KUKA KRL program: MyProgram_180().src

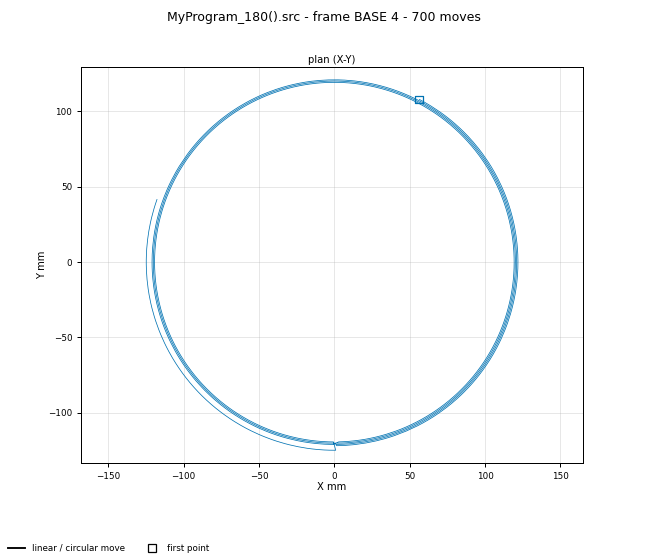
[picture p0: tool path of MyProgram_180().src in frame BASE 4, 700 of 700 moves have a stored position in this frame; points joined in program order, loops and branches not executed]
&ACCESS RVP
&REL 1
&PARAM TEMPLATE = C:\KRC\Roboter\Template\vorgabe
&PARAM EDITMASK = *
DEF MyProgram_180()
; ---- Setting reference (Base) ----
$BASE = BASE_DATA[4]

; --------------------------
; ---- Setting tool (TCP) ----
$TOOL = TOOL_DATA[3]
; --------------------------

$VEL.CP = VEL_APROX_PRINT
Startdeposition()
$VEL.CP = VEL_PRINT
LIN {X 56.4731,Y 107.9839,Z 132,A 57.7826,B 24.9435,C -1.7366,E1 25.0755,E2 388.3875} C_DIS
LIN {X 60.1294,Y 105.9923,Z 132,A 56.1238,B 24.9427,C -1.7481,E1 25.0795,E2 390.0143} C_DIS
LIN {X 64.0212,Y 103.6878,Z 132,A 53.6842,B 24.9439,C -1.7299,E1 25.0854,E2 392.4894} C_DIS
LIN {X 70.1878,Y 99.6172,Z 132,A 50.2313,B 24.9442,C -1.7251,E1 25.0934,E2 395.942} C_DIS
LIN {X 73.4213,Y 97.2579,Z 132,A 48.296,B 24.9446,C -1.7192,E1 25.0977,E2 397.8843} C_DIS
LIN {X 77.0237,Y 94.4306,Z 132,A 46.2185,B 24.9446,C -1.7188,E1 25.1023,E2 399.9551} C_DIS
LIN {X 80.294,Y 91.6663,Z 132,A 44.3805,B 24.9443,C -1.7233,E1 25.1061,E2 401.7753} C_DIS
LIN {X 83.0267,Y 89.1984,Z 132,A 42.6386,B 24.9446,C -1.7192,E1 25.1097,E2 403.5198} C_DIS
LIN {X 85.7566,Y 86.578,Z 132,A 40.7263,B 24.9453,C -1.7089,E1 25.1136,E2 405.4483} C_DIS
LIN {X 88.8179,Y 83.4346,Z 132,A 38.6725,B 24.9455,C -1.7048,E1 25.1175,E2 407.5031} C_DIS
LIN {X 92.0346,Y 79.8719,Z 132,A 36.4485,B 24.9458,C -1.7012,E1 25.1217,E2 409.7257} C_DIS
LIN {X 95.6699,Y 75.4792,Z 132,A 33.745,B 24.9462,C -1.6936,E1 25.1264,E2 412.4344} C_DIS
LIN {X 98.202,Y 72.1549,Z 132,A 31.8136,B 24.9465,C -1.6903,E1 25.1297,E2 414.3644} C_DIS
LIN {X 102.2261,Y 66.3297,Z 132,A 28.5147,B 24.9469,C -1.6831,E1 25.1349,E2 417.664} C_DIS
LIN {X 104.0153,Y 63.4873,Z 132,A 26.4897,B 24.9485,C -1.6571,E1 25.1379,E2 419.7401} C_DIS
LIN {X 106.1427,Y 59.8631,Z 132,A 24.9613,B 24.9475,C -1.6736,E1 25.1399,E2 421.2217} C_DIS
LIN {X 108.2856,Y 55.8944,Z 132,A 22.9017,B 24.9477,C -1.6706,E1 25.1426,E2 423.2774} C_DIS
LIN {X 110.9683,Y 50.3551,Z 132,A 20.0051,B 24.9482,C -1.6622,E1 25.1461,E2 426.1783} C_DIS
LIN {X 112.7882,Y 46.1367,Z 132,A 17.4555,B 24.9498,C -1.6366,E1 25.1489,E2 428.774} C_DIS
LIN {X 114.2155,Y 42.4817,Z 132,A 15.9852,B 24.949,C -1.6496,E1 25.1503,E2 430.2057} C_DIS
LIN {X 115.6712,Y 38.3389,Z 132,A 13.9725,B 24.9492,C -1.6459,E1 25.1521,E2 432.2157} C_DIS
LIN {X 116.887,Y 34.4575,Z 132,A 11.9721,B 24.9499,C -1.6356,E1 25.1537,E2 434.2289} C_DIS
LIN {X 118.1425,Y 29.8669,Z 132,A 9.3487,B 24.9515,C -1.6096,E1 25.1556,E2 436.8985} C_DIS
LIN {X 119.1512,Y 25.5527,Z 132,A 7.3765,B 24.9515,C -1.6085,E1 25.1568,E2 438.8619} C_DIS
LIN {X 119.9017,Y 21.7572,Z 132,A 5.7778,B 24.9512,C -1.6136,E1 25.1576,E2 440.4392} C_DIS
LIN {X 120.553,Y 17.8008,Z 132,A 3.3375,B 24.9532,C -1.5801,E1 25.1586,E2 442.944} C_DIS
LIN {X 121.2462,Y 12.2184,Z 132,A 0.9458,B 24.953,C -1.584,E1 25.1592,E2 445.3124} C_DIS
LIN {X 121.6093,Y 7.7983,Z 132,A -0.5381,B 24.9516,C -1.6071,E1 25.1595,E2 446.7331} C_DIS
LIN {X 121.7541,Y 5.0713,Z 132,A -2.4124,B 24.9536,C -1.5735,E1 25.1598,E2 448.6753} C_DIS
LIN {X 121.8578,Y 0.5482,Z 132,A -3.7742,B 24.9518,C -1.6047,E1 25.1598,E2 449.9557} C_DIS
LIN {X 121.787,Y -4.1979,Z 132,A -6.1962,B 24.9528,C -1.5878,E1 25.1597,E2 452.4031} C_DIS
LIN {X 121.5815,Y -8.2299,Z 132,A -8.1191,B 24.9532,C -1.5803,E1 25.1593,E2 454.3322} C_DIS
LIN {X 121.104,Y -13.5503,Z 132,A -11.226,B 24.9554,C -1.5425,E1 25.1584,E2 457.5097} C_DIS
LIN {X 120.4386,Y -18.5544,Z 132,A -12.6686,B 24.9532,C -1.5811,E1 25.1579,E2 458.853} C_DIS
LIN {X 119.981,Y -21.319,Z 132,A -14.6634,B 24.9554,C -1.5429,E1 25.1569,E2 460.9259} C_DIS
LIN {X 119.1633,Y -25.4976,Z 132,A -16.7801,B 24.9561,C -1.5307,E1 25.1556,E2 463.0591} C_DIS
LIN {X 118.136,Y -29.8926,Z 132,A -18.3594,B 24.9549,C -1.5509,E1 25.1546,E2 464.5818} C_DIS
LIN {X 116.8997,Y -34.4146,Z 132,A -21.4806,B 24.9579,C -1.4984,E1 25.1521,E2 467.8089} C_DIS
LIN {X 114.889,Y -40.6276,Z 132,A -23.6416,B 24.9559,C -1.5336,E1 25.1502,E2 469.8748} C_DIS
LIN {X 113.2694,Y -44.9444,Z 132,A -25.6739,B 24.9559,C -1.5336,E1 25.1482,E2 471.8959} C_DIS
LIN {X 110.7217,Y -50.8989,Z 132,A -28.8215,B 24.9568,C -1.519,E1 25.1446,E2 475.0605} C_DIS
LIN {X 109.2594,Y -53.9659,Z 132,A -30.6777,B 24.9578,C -1.5013,E1 25.1423,E2 476.9486} C_DIS
LIN {X 107.6556,Y -57.0968,Z 132,A -32.5414,B 24.9586,C -1.486,E1 25.1398,E2 478.8386} C_DIS
LIN {X 105.4079,Y -61.1478,Z 132,A -34.1894,B 24.9575,C -1.5057,E1 25.1376,E2 480.4314} C_DIS
LIN {X 103.2812,Y -64.676,Z 132,A -36.1228,B 24.9578,C -1.5003,E1 25.1348,E2 482.3679} C_DIS
LIN {X 100.9382,Y -68.274,Z 132,A -38.0879,B 24.958,C -1.4972,E1 25.1318,E2 484.3305} C_DIS
LIN {X 98.55,Y -71.6776,Z 132,A -40.0435,B 24.9583,C -1.4917,E1 25.1286,E2 486.2896} C_DIS
LIN {X 96.0385,Y -75.0101,Z 132,A -42.2663,B 24.9593,C -1.4734,E1 25.1247,E2 488.545} C_DIS
LIN {X 93.9447,Y -77.6163,Z 132,A -43.566,B 24.9588,C -1.4826,E1 25.1225,E2 489.8168} C_DIS
LIN {X 91.9011,Y -80.0264,Z 132,A -45.4055,B 24.96,C -1.4613,E1 25.1191,E2 491.6985} C_DIS
LIN {X 89.3899,Y -82.8206,Z 132,A -47.373,B 24.9608,C -1.4469,E1 25.1153,E2 493.6911} C_DIS
LIN {X 86.0477,Y -86.2879,Z 132,A -49.0581,B 24.9595,C -1.4697,E1 25.1121,E2 495.3154} C_DIS
LIN {X 83.8181,Y -88.4552,Z 132,A -50.9541,B 24.9609,C -1.4448,E1 25.1081,E2 497.2622} C_DIS
LIN {X 80.6989,Y -91.31,Z 132,A -52.893,B 24.961,C -1.4426,E1 25.1041,E2 499.1988} C_DIS
LIN {X 77.6217,Y -93.9402,Z 132,A -54.3862,B 24.9602,C -1.4583,E1 25.101,E2 500.6491} C_DIS
LIN {X 74.3584,Y -96.5433,Z 132,A -57.188,B 24.9626,C -1.4132,E1 25.0946,E2 503.547} C_DIS
LIN {X 69.3835,Y -100.1788,Z 132,A -59.2103,B 24.9606,C -1.4496,E1 25.0902,E2 505.4765} C_DIS
LIN {X 66.0306,Y -102.4196,Z 132,A -61.1258,B 24.9609,C -1.4449,E1 25.0857,E2 507.3968} C_DIS
LIN {X 62.3586,Y -104.6957,Z 132,A -63.1483,B 24.9611,C -1.4414,E1 25.0808,E2 509.4211} C_DIS
LIN {X 58.664,Y -106.8099,Z 132,A -65.125,B 24.9612,C -1.439,E1 25.076,E2 511.3977} C_DIS
LIN {X 55.147,Y -108.6664,Z 132,A -66.7851,B 24.9608,C -1.446,E1 25.072,E2 513.0367} C_DIS
LIN {X 47.6474,Y -112.1587,Z 132,A -70.8114,B 24.9615,C -1.4332,E1 25.0617,E2 517.083} C_DIS
LIN {X 39.8361,Y -115.1649,Z 132,A -74.7717,B 24.9619,C -1.4265,E1 25.0513,E2 521.0506} C_DIS
LIN {X 35.9115,Y -116.4481,Z 132,A -76.6767,B 24.9619,C -1.4259,E1 25.0463,E2 522.9535} C_DIS
LIN {X 33.0929,Y -117.2805,Z 132,A -78.8349,B 24.9639,C -1.3875,E1 25.0402,E2 525.1992} C_DIS
LIN {X 27.7021,Y -118.6696,Z 132,A -80.6741,B 24.9621,C -1.4217,E1 25.0355,E2 526.9546} C_DIS
LIN {X 20.9444,Y -120.0462,Z 132,A -83.8401,B 24.9621,C -1.4226,E1 25.0268,E2 530.1149} C_DIS
LIN {X 13.1586,Y -121.1476,Z 132,A -87.6463,B 24.9625,C -1.4149,E1 25.0162,E2 533.936} C_DIS
LIN {X 7.5514,Y -121.625,Z 132,A -90.2781,B 24.9625,C -1.4143,E1 25.0089,E2 536.568} C_DIS
LIN {X 1.6031,Y -121.8492,Z 132,A -93.0648,B 24.9625,C -1.4139,E1 25.0011,E2 539.3549} C_DIS
LIN {X 1.6031,Y -121.8492,Z 132,A -93.0648,B 24.9625,C -1.4139,E1 25.0011,E2 539.3549} C_DIS
Enddeposition()
LIN {X 0.8619,Y -121.0153,Z 132,A -93.2429,B 24.9613,C -1.4367,E1 25.0008,E2 539.4791} C_DIS
Startdeposition()
$VEL.CP = VEL_PRINT
LIN {X 6.3359,Y -120.8553,Z 132,A -90.2443,B 24.9603,C -1.4565,E1 25.0093,E2 536.4343} C_DIS
LIN {X 11.7186,Y -120.4527,Z 132,A -87.5229,B 24.9598,C -1.4656,E1 25.0169,E2 533.6928} C_DIS
LIN {X 19.5929,Y -119.4252,Z 132,A -83.8748,B 24.9599,C -1.4627,E1 25.027,E2 530.0546} C_DIS
LIN {X 25.3127,Y -118.3457,Z 132,A -80.8984,B 24.9592,C -1.4756,E1 25.0352,E2 527.0512} C_DIS
LIN {X 29.533,Y -117.3621,Z 132,A -78.4741,B 24.9581,C -1.4957,E1 25.0419,E2 524.5829} C_DIS
LIN {X 33.3995,Y -116.3213,Z 132,A -77.3045,B 24.9599,C -1.4627,E1 25.0448,E2 523.4933} C_DIS
LIN {X 36.2161,Y -115.4764,Z 132,A -75.5363,B 24.9588,C -1.4824,E1 25.0496,E2 521.6815} C_DIS
LIN {X 40.4165,Y -114.0742,Z 132,A -72.6762,B 24.9566,C -1.5225,E1 25.0574,E2 518.7324} C_DIS
LIN {X 45.9816,Y -111.946,Z 132,A -71.087,B 24.9597,C -1.4664,E1 25.0612,E2 517.2796} C_DIS
LIN {X 48.5992,Y -110.8351,Z 132,A -68.8991,B 24.9573,C -1.5094,E1 25.067,E2 514.9952} C_DIS
LIN {X 52.3751,Y -109.1004,Z 132,A -67.3976,B 24.9584,C -1.4898,E1 25.0707,E2 513.544} C_DIS
LIN {X 55.1873,Y -107.7059,Z 132,A -65.894,B 24.9582,C -1.4931,E1 25.0744,E2 512.0366} C_DIS
LIN {X 58.9166,Y -105.7121,Z 132,A -63.956,B 24.9582,C -1.4935,E1 25.0792,E2 510.1032} C_DIS
LIN {X 62.4253,Y -103.6791,Z 132,A -62.0096,B 24.9579,C -1.4984,E1 25.0839,E2 508.1513} C_DIS
LIN {X 65.9772,Y -101.4559,Z 132,A -60.0117,B 24.9577,C -1.503,E1 25.0886,E2 506.149} C_DIS
LIN {X 69.5361,Y -99.0503,Z 132,A -57.5135,B 24.9561,C -1.5302,E1 25.0944,E2 503.5952} C_DIS
LIN {X 73.0802,Y -96.465,Z 132,A -56.2087,B 24.958,C -1.4964,E1 25.0972,E2 502.3748} C_DIS
LIN {X 75.3002,Y -94.7432,Z 132,A -54.6377,B 24.9572,C -1.5112,E1 25.1007,E2 500.7747} C_DIS
LIN {X 78.4324,Y -92.1664,Z 132,A -52.4997,B 24.9563,C -1.5264,E1 25.1053,E2 498.6091} C_DIS
LIN {X 82.7817,Y -88.2817,Z 132,A -49.9854,B 24.9567,C -1.5207,E1 25.1104,E2 496.1184} C_DIS
LIN {X 85.5435,Y -85.6068,Z 132,A -48.159,B 24.9564,C -1.5255,E1 25.1141,E2 494.2883} C_DIS
LIN {X 89.2906,Y -81.691,Z 132,A -45.4198,B 24.9555,C -1.5407,E1 25.1194,E2 491.5252} C_DIS
LIN {X 92.6227,Y -77.8929,Z 132,A -43.2156,B 24.9557,C -1.5376,E1 25.1233,E2 489.3384} C_DIS
LIN {X 95.544,Y -74.2806,Z 132,A -41.0799,B 24.9555,C -1.5404,E1 25.127,E2 487.2061} C_DIS
LIN {X 97.8502,Y -71.2148,Z 132,A -39.2128,B 24.9551,C -1.548,E1 25.1302,E2 485.3301} C_DIS
LIN {X 100.1998,Y -67.87,Z 132,A -37.2787,B 24.9548,C -1.5534,E1 25.1332,E2 483.3927} C_DIS
LIN {X 102.5089,Y -64.3297,Z 132,A -35.3029,B 24.9545,C -1.5579,E1 25.1362,E2 481.4163} C_DIS
LIN {X 104.6427,Y -60.796,Z 132,A -33.1046,B 24.9535,C -1.5759,E1 25.1394,E2 479.1868} C_DIS
LIN {X 106.2599,Y -57.9229,Z 132,A -31.7333,B 24.9538,C -1.571,E1 25.1412,E2 477.8342} C_DIS
LIN {X 108.1595,Y -54.2924,Z 132,A -29.9502,B 24.9538,C -1.569,E1 25.1434,E2 476.0653} C_DIS
LIN {X 109.8398,Y -50.8089,Z 132,A -28.0388,B 24.9533,C -1.5786,E1 25.1457,E2 474.1415} C_DIS
LIN {X 112.2274,Y -45.2912,Z 132,A -25.4363,B 24.9535,C -1.5752,E1 25.1485,E2 471.5613} C_DIS
LIN {X 113.4229,Y -42.2084,Z 132,A -23.6268,B 24.9525,C -1.5924,E1 25.1503,E2 469.7215} C_DIS
LIN {X 115.6424,Y -35.6797,Z 132,A -20.661,B 24.9528,C -1.5877,E1 25.153,E2 466.7834} C_DIS
LIN {X 116.5793,Y -32.4882,Z 132,A -18.8947,B 24.9519,C -1.6024,E1 25.1543,E2 464.9926} C_DIS
LIN {X 117.5779,Y -28.6609,Z 132,A -16.8322,B 24.9509,C -1.618,E1 25.1557,E2 462.9051} C_DIS
LIN {X 118.605,Y -24.0629,Z 132,A -14.249,B 24.9494,C -1.6432,E1 25.1572,E2 460.2778} C_DIS
LIN {X 119.4497,Y -19.4417,Z 132,A -12.6063,B 24.9508,C -1.621,E1 25.1579,E2 458.6971} C_DIS
LIN {X 120.0419,Y -15.3706,Z 132,A -10.5678,B 24.9501,C -1.6319,E1 25.1587,E2 456.6447} C_DIS
LIN {X 120.6869,Y -9.0042,Z 132,A -7.7119,B 24.9501,C -1.6331,E1 25.1594,E2 453.803} C_DIS
LIN {X 120.9011,Y -5.4111,Z 132,A -5.2894,B 24.9474,C -1.6751,E1 25.1598,E2 451.296} C_DIS
LIN {X 121.0219,Y -0.1787,Z 132,A -3.7488,B 24.9499,C -1.6358,E1 25.1598,E2 449.8571} C_DIS
LIN {X 120.855,Y 6.3424,Z 132,A -0.7721,B 24.9496,C -1.6402,E1 25.1596,E2 446.8877} C_DIS
LIN {X 120.334,Y 12.882,Z 132,A 2.4886,B 24.9485,C -1.658,E1 25.1588,E2 443.6045} C_DIS
LIN {X 119.5793,Y 18.6237,Z 132,A 5.3509,B 24.9476,C -1.6728,E1 25.1577,E2 440.7241} C_DIS
LIN {X 118.1469,Y 26.22,Z 132,A 9.188,B 24.9463,C -1.6932,E1 25.1556,E2 436.8611} C_DIS
LIN {X 117.078,Y 30.641,Z 132,A 11.1547,B 24.9464,C -1.6906,E1 25.1542,E2 434.912} C_DIS
LIN {X 115.9402,Y 34.7003,Z 132,A 13.141,B 24.9461,C -1.6963,E1 25.1527,E2 432.9237} C_DIS
LIN {X 114.6407,Y 38.7777,Z 132,A 15.1666,B 24.9457,C -1.7024,E1 25.1509,E2 430.895} C_DIS
LIN {X 113.1995,Y 42.8013,Z 132,A 17.6033,B 24.944,C -1.7292,E1 25.1485,E2 428.4088} C_DIS
LIN {X 111.6487,Y 46.6989,Z 132,A 19.1155,B 24.9451,C -1.7113,E1 25.1469,E2 426.947} C_DIS
LIN {X 108.2803,Y 54.0518,Z 132,A 22.7188,B 24.9451,C -1.7111,E1 25.1427,E2 423.3639} C_DIS
LIN {X 106.0847,Y 58.2432,Z 132,A 25.1799,B 24.944,C -1.7283,E1 25.1394,E2 420.8751} C_DIS
LIN {X 102.1993,Y 64.8191,Z 132,A 29.6095,B 24.9407,C -1.7785,E1 25.1328,E2 416.3495} C_DIS
LIN {X 98.8039,Y 69.887,Z 132,A 31.6432,B 24.943,C -1.7434,E1 25.1297,E2 414.4086} C_DIS
LIN {X 96.3363,Y 73.25,Z 132,A 33.6242,B 24.9427,C -1.7487,E1 25.1264,E2 412.4248} C_DIS
LIN {X 93.2695,Y 77.1172,Z 132,A 36.0737,B 24.942,C -1.7599,E1 25.1221,E2 409.9602} C_DIS
LIN {X 90.9591,Y 79.8289,Z 132,A 37.556,B 24.9424,C -1.7538,E1 25.1194,E2 408.4989} C_DIS
LIN {X 88.404,Y 82.6504,Z 132,A 39.3861,B 24.942,C -1.7592,E1 25.1159,E2 406.664} C_DIS
LIN {X 85.5476,Y 85.6026,Z 132,A 41.3288,B 24.9417,C -1.7634,E1 25.1121,E2 404.7198} C_DIS
LIN {X 82.1623,Y 88.8575,Z 132,A 43.381,B 24.942,C -1.7597,E1 25.108,E2 402.6848} C_DIS
LIN {X 79.5084,Y 91.2409,Z 132,A 45.2342,B 24.9412,C -1.7711,E1 25.1041,E2 400.812} C_DIS
LIN {X 76.4254,Y 93.837,Z 132,A 47.1191,B 24.941,C -1.7737,E1 25.1,E2 398.9283} C_DIS
LIN {X 73.1083,Y 96.4438,Z 132,A 48.9233,B 24.9414,C -1.768,E1 25.0961,E2 397.144} C_DIS
LIN {X 70.4757,Y 98.3841,Z 132,A 50.6238,B 24.9407,C -1.7781,E1 25.0922,E2 395.4257} C_DIS
LIN {X 65.4847,Y 101.7742,Z 132,A 53.3213,B 24.9409,C -1.7751,E1 25.086,E2 392.7442} C_DIS
LIN {X 62.7738,Y 103.4683,Z 132,A 55.3392,B 24.9392,C -1.8018,E1 25.081,E2 390.6697} C_DIS
LIN {X 59.6414,Y 105.3056,Z 132,A 56.6863,B 24.9402,C -1.7863,E1 25.0779,E2 389.3631} C_DIS
LIN {X 56.2147,Y 107.1732,Z 132,A 58.5668,B 24.9399,C -1.7904,E1 25.0732,E2 387.4782} C_DIS
LIN {X 52.7332,Y 108.9284,Z 132,A 60.735,B 24.9387,C -1.8082,E1 25.0677,E2 385.2738} C_DIS
LIN {X 49.5239,Y 110.4238,Z 132,A 62.009,B 24.9399,C -1.7909,E1 25.0646,E2 384.0439} C_DIS
LIN {X 46.1664,Y 111.8699,Z 132,A 64.21,B 24.9382,C -1.8152,E1 25.0588,E2 381.7905} C_DIS
LIN {X 42.5085,Y 113.3102,Z 132,A 65.6592,B 24.9394,C -1.7974,E1 25.0551,E2 380.3866} C_DIS
LIN {X 38.5616,Y 114.7138,Z 132,A 67.6786,B 24.9392,C -1.8009,E1 25.0498,E2 378.3631} C_DIS
LIN {X 34.2989,Y 116.0597,Z 132,A 69.7886,B 24.9392,C -1.8022,E1 25.0441,E2 376.2537} C_DIS
LIN {X 30.263,Y 117.1766,Z 132,A 71.7559,B 24.9391,C -1.8028,E1 25.0388,E2 374.2881} C_DIS
LIN {X 26.0692,Y 118.1805,Z 132,A 74.292,B 24.9374,C -1.8272,E1 25.0318,E2 371.6976} C_DIS
LIN {X 21.688,Y 119.0624,Z 132,A 75.8305,B 24.9392,C -1.8009,E1 25.0277,E2 370.2232} C_DIS
LIN {X 18.0785,Y 119.6638,Z 132,A 77.6555,B 24.9389,C -1.8057,E1 25.0227,E2 368.3883} C_DIS
LIN {X 13.143,Y 120.3061,Z 132,A 80.3298,B 24.9378,C -1.821,E1 25.0151,E2 365.6798} C_DIS
LIN {X 9.4835,Y 120.6494,Z 132,A 81.2967,B 24.9403,C -1.7853,E1 25.0127,E2 364.7982} C_DIS
LIN {X 6.8629,Y 120.8273,Z 132,A 83.4794,B 24.9373,C -1.8288,E1 25.0063,E2 362.5131} C_DIS
LIN {X 2.3958,Y 120.9981,Z 132,A 85.3236,B 24.9382,C -1.8159,E1 25.0013,E2 360.6999} C_DIS
LIN {X -3.8709,Y 120.9593,Z 132,A 87.8709,B 24.9396,C -1.7958,E1 24.9943,E2 358.2002} C_DIS
LIN {X -9.7792,Y 120.6252,Z 132,A 90.6844,B 24.9396,C -1.7952,E1 24.9865,E2 355.3872} C_DIS
LIN {X -15.3027,Y 120.0504,Z 132,A 93.4972,B 24.9391,C -1.802,E1 24.9786,E2 352.5563} C_DIS
LIN {X -19.2992,Y 119.4728,Z 132,A 95.7723,B 24.9381,C -1.8173,E1 24.9722,E2 350.2428} C_DIS
LIN {X -23.0037,Y 118.8146,Z 132,A 97.0951,B 24.9396,C -1.795,E1 24.9687,E2 348.9717} C_DIS
LIN {X -27.2474,Y 117.9143,Z 132,A 98.9117,B 24.9405,C -1.7824,E1 24.9638,E2 347.1827} C_DIS
LIN {X -30.0462,Y 117.2326,Z 132,A 100.6466,B 24.9394,C -1.7978,E1 24.959,E2 345.4087} C_DIS
LIN {X -34.2834,Y 116.0643,Z 132,A 102.7357,B 24.9395,C -1.7959,E1 24.9534,E2 343.3208} C_DIS
LIN {X -38.444,Y 114.7536,Z 132,A 104.7629,B 24.9398,C -1.7917,E1 24.9481,E2 341.2998} C_DIS
LIN {X -44.5466,Y 112.5259,Z 132,A 107.9094,B 24.9398,C -1.7908,E1 24.9398,E2 338.1491} C_DIS
LIN {X -48.248,Y 110.988,Z 132,A 109.7153,B 24.9404,C -1.7839,E1 24.9352,E2 336.3552} C_DIS
LIN {X -51.4904,Y 109.522,Z 132,A 111.4881,B 24.9403,C -1.7852,E1 24.9307,E2 334.575} C_DIS
LIN {X -55.5598,Y 107.5153,Z 132,A 113.4775,B 24.941,C -1.7746,E1 24.9258,E2 332.6055} C_DIS
LIN {X -58.506,Y 105.9409,Z 132,A 115.217,B 24.9407,C -1.7789,E1 24.9215,E2 330.8509} C_DIS
LIN {X -63.4121,Y 103.0776,Z 132,A 117.9733,B 24.9408,C -1.7769,E1 24.9149,E2 328.0909} C_DIS
LIN {X -67.4091,Y 100.5101,Z 132,A 120.1331,B 24.9414,C -1.7685,E1 24.9099,E2 325.9439} C_DIS
LIN {X -70.7451,Y 98.1913,Z 132,A 122.0973,B 24.9415,C -1.7664,E1 24.9054,E2 323.9781} C_DIS
LIN {X -74.1916,Y 95.613,Z 132,A 124.1357,B 24.9418,C -1.7621,E1 24.9009,E2 321.9426} C_DIS
LIN {X -77.4323,Y 93.0078,Z 132,A 126.1221,B 24.942,C -1.7585,E1 24.8966,E2 319.9572} C_DIS
LIN {X -80.6687,Y 90.2151,Z 132,A 128.1497,B 24.9423,C -1.754,E1 24.8923,E2 317.9323} C_DIS
LIN {X -83.7677,Y 87.3457,Z 132,A 130.1541,B 24.9426,C -1.7494,E1 24.8883,E2 315.9306} C_DIS
LIN {X -86.7948,Y 84.3384,Z 132,A 132.1754,B 24.943,C -1.7445,E1 24.8843,E2 313.9125} C_DIS
LIN {X -89.5933,Y 81.3592,Z 132,A 134.1427,B 24.9432,C -1.741,E1 24.8806,E2 311.9448} C_DIS
LIN {X -92.3797,Y 78.1805,Z 132,A 136.1442,B 24.9435,C -1.7358,E1 24.8769,E2 309.9466} C_DIS
LIN {X -95.0184,Y 74.9517,Z 132,A 138.1334,B 24.9438,C -1.7311,E1 24.8735,E2 307.9591} C_DIS
LIN {X -97.5212,Y 71.6659,Z 132,A 140.1309,B 24.9441,C -1.7276,E1 24.8701,E2 305.9605} C_DIS
LIN {X -102.9065,Y 63.6906,Z 132,A 144.1689,B 24.9463,C -1.6922,E1 24.864,E2 301.9867} C_DIS
LIN {X -105.1169,Y 59.9721,Z 132,A 147.6673,B 24.9427,C -1.7492,E1 24.8589,E2 298.3341} C_DIS
LIN {X -108.1317,Y 54.3472,Z 132,A 149.6399,B 24.9462,C -1.6944,E1 24.8565,E2 296.4817} C_DIS
LIN {X -109.6964,Y 51.1166,Z 132,A 151.4702,B 24.9462,C -1.6949,E1 24.8543,E2 294.6403} C_DIS
LIN {X -111.2663,Y 47.6013,Z 132,A 153.4384,B 24.9462,C -1.6955,E1 24.8521,E2 292.6596} C_DIS
LIN {X -113.0721,Y 43.1386,Z 132,A 155.6056,B 24.9469,C -1.6836,E1 24.8499,E2 290.5088} C_DIS
LIN {X -114.5689,Y 38.9884,Z 132,A 158.0775,B 24.9463,C -1.6936,E1 24.8476,E2 287.9991} C_DIS
LIN {X -115.7125,Y 35.4503,Z 132,A 159.2285,B 24.9483,C -1.6617,E1 24.8467,E2 286.9175} C_DIS
LIN {X -116.592,Y 32.4425,Z 132,A 160.9841,B 24.9478,C -1.6686,E1 24.8453,E2 285.1352} C_DIS
LIN {X -117.6861,Y 28.2168,Z 132,A 163.0967,B 24.9481,C -1.6639,E1 24.8439,E2 283.0214} C_DIS
LIN {X -118.5744,Y 24.2115,Z 132,A 164.967,B 24.9487,C -1.6545,E1 24.8428,E2 281.1625} C_DIS
LIN {X -119.2676,Y 20.528,Z 132,A 166.8096,B 24.9489,C -1.6517,E1 24.8419,E2 279.3158} C_DIS
LIN {X -119.884,Y 16.5541,Z 132,A 168.7107,B 24.9493,C -1.6453,E1 24.8411,E2 277.4185} C_DIS
LIN {X -120.632,Y 9.6961,Z 132,A 171.6014,B 24.9509,C -1.6185,E1 24.8403,E2 274.5744} C_DIS
LIN {X -120.912,Y 5.1493,Z 132,A 174.4229,B 24.9496,C -1.64,E1 24.8399,E2 271.6847} C_DIS
LIN {X -121.0227,Y 0.0056,Z 132,A 176.9017,B 24.95,C -1.6339,E1 24.8399,E2 269.2056} C_DIS
LIN {X -120.9795,Y -3.2147,Z 132,A 178.0867,B 24.9512,C -1.6142,E1 24.8399,E2 268.0603} C_DIS
LIN {X -120.8505,Y -6.4289,Z 132,A 179.6443,B 24.9514,C -1.6108,E1 24.8401,E2 266.5015} C_DIS
LIN {X -120.5912,Y -10.193,Z 132,A -178.3971,B 24.9513,C -1.6124,E1 24.8405,E2 264.5272} C_DIS
LIN {X -120.0638,Y -15.1959,Z 132,A -176.0666,B 24.9519,C -1.6025,E1 24.8413,E2 262.2064} C_DIS
LIN {X -119.4793,Y -19.2593,Z 132,A -174.149,B 24.9523,C -1.5952,E1 24.8421,E2 260.2949} C_DIS
LIN {X -118.7708,Y -23.2302,Z 132,A -172.1998,B 24.9526,C -1.5908,E1 24.8431,E2 258.3445} C_DIS
LIN {X -117.8088,Y -27.703,Z 132,A -169.9737,B 24.9528,C -1.5866,E1 24.8444,E2 256.1153} C_DIS
LIN {X -116.7331,Y -31.9346,Z 132,A -167.9257,B 24.9533,C -1.5793,E1 24.8459,E2 254.0728} C_DIS
LIN {X -115.5368,Y -36.0229,Z 132,A -165.3999,B 24.9523,C -1.5954,E1 24.848,E2 251.4942} C_DIS
LIN {X -114.1241,Y -40.2754,Z 132,A -163.9666,B 24.9545,C -1.5589,E1 24.8493,E2 250.1396} C_DIS
LIN {X -112.7368,Y -44.0069,Z 132,A -162.1829,B 24.9551,C -1.5489,E1 24.851,E2 248.3698} C_DIS
LIN {X -111.7199,Y -46.5299,Z 132,A -160.5601,B 24.9544,C -1.5597,E1 24.8527,E2 246.7122} C_DIS
LIN {X -109.9083,Y -50.662,Z 132,A -158.6584,B 24.9554,C -1.5433,E1 24.8549,E2 244.8392} C_DIS
LIN {X -108.5856,Y -53.4358,Z 132,A -156.9325,B 24.9549,C -1.551,E1 24.857,E2 243.0856} C_DIS
LIN {X -105.5833,Y -59.1471,Z 132,A -154.2085,B 24.9563,C -1.528,E1 24.8606,E2 240.4019} C_DIS
LIN {X -104.1987,Y -61.5547,Z 132,A -152.6144,B 24.9558,C -1.5366,E1 24.8628,E2 238.779} C_DIS
LIN {X -102.1852,Y -64.8413,Z 132,A -150.7866,B 24.956,C -1.5319,E1 24.8655,E2 236.9532} C_DIS
LIN {X -100.3931,Y -67.5828,Z 132,A -149.1702,B 24.956,C -1.5308,E1 24.868,E2 235.3314} C_DIS
LIN {X -97.9457,Y -71.0837,Z 132,A -146.8831,B 24.9557,C -1.5373,E1 24.8718,E2 233.0174} C_DIS
LIN {X -95.9568,Y -73.7464,Z 132,A -145.2325,B 24.9557,C -1.5369,E1 24.8746,E2 231.36} C_DIS
LIN {X -93.6968,Y -76.5972,Z 132,A -144.0467,B 24.9573,C -1.509,E1 24.8766,E2 230.2352} C_DIS
LIN {X -91.6114,Y -79.0795,Z 132,A -142.298,B 24.957,C -1.5148,E1 24.8798,E2 228.4645} C_DIS
LIN {X -87.9265,Y -83.1573,Z 132,A -140.0309,B 24.9582,C -1.4941,E1 24.884,E2 226.2367} C_DIS
LIN {X -86.0588,Y -85.0894,Z 132,A -137.6608,B 24.9555,C -1.5404,E1 24.8889,E2 223.7463} C_DIS
LIN {X -82.0702,Y -88.943,Z 132,A -135.9402,B 24.9582,C -1.4943,E1 24.8922,E2 222.1285} C_DIS
LIN {X -79.494,Y -91.2534,Z 132,A -133.9901,B 24.9576,C -1.5049,E1 24.8964,E2 220.1453} C_DIS
LIN {X -75.2252,Y -94.8027,Z 132,A -131.5963,B 24.9584,C -1.4894,E1 24.9015,E2 217.7794} C_DIS
LIN {X -72.3478,Y -97.0159,Z 132,A -129.307,B 24.9572,C -1.5121,E1 24.9067,E2 215.4278} C_DIS
LIN {X -68.9718,Y -99.4442,Z 132,A -127.9183,B 24.9588,C -1.4825,E1 24.9098,E2 214.1047} C_DIS
LIN {X -65.9796,Y -101.4543,Z 132,A -126.1183,B 24.9588,C -1.484,E1 24.914,E2 212.2953} C_DIS
LIN {X -62.1675,Y -103.8339,Z 132,A -124.2286,B 24.9595,C -1.47,E1 24.9184,E2 210.433} C_DIS
LIN {X -59.6592,Y -105.2956,Z 132,A -122.5433,B 24.9588,C -1.4821,E1 24.9225,E2 208.714} C_DIS
LIN {X -56.042,Y -107.2635,Z 132,A -120.3228,B 24.9583,C -1.4919,E1 24.9281,E2 206.464} C_DIS
LIN {X -53.0337,Y -108.7825,Z 132,A -119.2117,B 24.9596,C -1.4678,E1 24.9308,E2 205.4074} C_DIS
LIN {X -50.2043,Y -110.117,Z 132,A -117.5032,B 24.9592,C -1.4764,E1 24.9351,E2 203.6741} C_DIS
LIN {X -45.1593,Y -112.2803,Z 132,A -115.2891,B 24.9603,C -1.4561,E1 24.9407,E2 201.5032} C_DIS
LIN {X -42.3874,Y -113.3559,Z 132,A -113.4937,B 24.9594,C -1.4725,E1 24.9455,E2 199.6651} C_DIS
LIN {X -38.5188,Y -114.7283,Z 132,A -111.5127,B 24.9594,C -1.4725,E1 24.9508,E2 197.68} C_DIS
LIN {X -34.5929,Y -115.9722,Z 132,A -109.5998,B 24.9596,C -1.4694,E1 24.9559,E2 195.7713} C_DIS
LIN {X -30.7386,Y -117.0522,Z 132,A -107.7528,B 24.9597,C -1.466,E1 24.9608,E2 193.9296} C_DIS
LIN {X -24.5347,Y -118.5078,Z 132,A -105.0759,B 24.9607,C -1.4487,E1 24.968,E2 191.2903} C_DIS
LIN {X -20.353,Y -119.2974,Z 132,A -102.6892,B 24.9598,C -1.4652,E1 24.9747,E2 188.8619} C_DIS
LIN {X -16.8673,Y -119.8398,Z 132,A -100.4386,B 24.9583,C -1.4921,E1 24.9811,E2 186.5457} C_DIS
LIN {X -12.169,Y -120.4089,Z 132,A -98.9887,B 24.9604,C -1.4546,E1 24.9849,E2 185.1839} C_DIS
LIN {X -6.3504,Y -120.8546,Z 132,A -96.324,B 24.9606,C -1.4499,E1 24.9923,E2 182.5292} C_DIS
LIN {X -0.7098,Y -121.0196,Z 132,A -93.3129,B 24.9597,C -1.4662,E1 25.0008,E2 179.4791} C_DIS
LIN {X -0.7098,Y -121.0196,Z 132,A -93.3129,B 24.9597,C -1.4662,E1 25.0008,E2 179.4791} C_DIS
Enddeposition()
LIN {X 0.8571,Y -120.1803,Z 132,A -93.1158,B 24.9603,C -1.4555,E1 25.0012,E2 179.3075} C_DIS
Startdeposition()
$VEL.CP = VEL_PRINT
LIN {X -4.0746,Y -120.1141,Z 132,A -95.6996,B 24.9609,C -1.4442,E1 24.994,E2 181.9181} C_DIS
LIN {X -8.9458,Y -119.8507,Z 132,A -98.2242,B 24.9614,C -1.435,E1 24.9869,E2 184.4654} C_DIS
LIN {X -12.6588,Y -119.5148,Z 132,A -100.0147,B 24.9614,C -1.4346,E1 24.9819,E2 186.2579} C_DIS
LIN {X -17.3508,Y -118.9244,Z 132,A -102.2021,B 24.9613,C -1.4381,E1 24.9758,E2 188.4386} C_DIS
LIN {X -21.4315,Y -118.257,Z 132,A -104.175,B 24.9613,C -1.4387,E1 24.9704,E2 190.4121} C_DIS
LIN {X -24.8804,Y -117.58,Z 132,A -105.9897,B 24.9615,C -1.4331,E1 24.9654,E2 192.2422} C_DIS
LIN {X -29.6231,Y -116.4754,Z 132,A -108.2154,B 24.9612,C -1.4387,E1 24.9594,E2 194.4576} C_DIS
LIN {X -33.9829,Y -115.2793,Z 132,A -110.347,B 24.9611,C -1.4412,E1 24.9537,E2 196.5867} C_DIS
LIN {X -37.9359,Y -114.039,Z 132,A -112.3131,B 24.961,C -1.4432,E1 24.9485,E2 198.5517} C_DIS
LIN {X -42.175,Y -112.5402,Z 132,A -114.3567,B 24.9606,C -1.4496,E1 24.9431,E2 200.5841} C_DIS
LIN {X -45.7083,Y -111.1521,Z 132,A -116.2672,B 24.9608,C -1.4469,E1 24.9381,E2 202.5052} C_DIS
LIN {X -49.0511,Y -109.7175,Z 132,A -117.8178,B 24.9602,C -1.457,E1 24.9342,E2 204.0355} C_DIS
LIN {X -52.2319,Y -108.2394,Z 132,A -119.5918,B 24.9604,C -1.4545,E1 24.9297,E2 205.82} C_DIS
LIN {X -55.5033,Y -106.5993,Z 132,A -121.449,B 24.9605,C -1.4517,E1 24.9251,E2 207.6888} C_DIS
LIN {X -59.2511,Y -104.5635,Z 132,A -123.4446,B 24.9603,C -1.4562,E1 24.9202,E2 209.6795} C_DIS
LIN {X -62.5304,Y -102.6353,Z 132,A -125.3077,B 24.9603,C -1.4567,E1 24.9157,E2 211.547} C_DIS
LIN {X -65.8349,Y -100.5485,Z 132,A -127.1926,B 24.9601,C -1.4587,E1 24.9113,E2 213.4334} C_DIS
LIN {X -69.4347,Y -98.0971,Z 132,A -129.2343,B 24.9599,C -1.4637,E1 24.9066,E2 215.4701} C_DIS
LIN {X -72.61,Y -95.7697,Z 132,A -131.154,B 24.9598,C -1.4651,E1 24.9023,E2 217.3932} C_DIS
LIN {X -76.0351,Y -93.0737,Z 132,A -133.1354,B 24.9593,C -1.4733,E1 24.898,E2 219.3627} C_DIS
LIN {X -78.7842,Y -90.7591,Z 132,A -134.9769,B 24.9595,C -1.471,E1 24.8941,E2 221.2168} C_DIS
LIN {X -81.3806,Y -88.4393,Z 132,A -137.1471,B 24.9605,C -1.4523,E1 24.8895,E2 223.4402} C_DIS
LIN {X -84.6717,Y -85.2932,Z 132,A -138.7783,B 24.959,C -1.4802,E1 24.8864,E2 225.0118} C_DIS
LIN {X -87.1093,Y -82.8012,Z 132,A -140.5906,B 24.9591,C -1.4774,E1 24.8829,E2 226.8387} C_DIS
LIN {X -90.3525,Y -79.2495,Z 132,A -142.7742,B 24.9586,C -1.4873,E1 24.8788,E2 229.0083} C_DIS
LIN {X -93.0594,Y -76.0527,Z 132,A -144.79,B 24.9583,C -1.4913,E1 24.8752,E2 231.0241} C_DIS
LIN {X -95.655,Y -72.7613,Z 132,A -146.454,B 24.9572,C -1.5106,E1 24.8724,E2 232.6499} C_DIS
LIN {X -97.4274,Y -70.3711,Z 132,A -148.2097,B 24.9579,C -1.4996,E1 24.8695,E2 234.4403} C_DIS
LIN {X -99.8147,Y -66.9411,Z 132,A -150.2009,B 24.9576,C -1.5048,E1 24.8663,E2 236.429} C_DIS
LIN {X -101.8216,Y -63.8478,Z 132,A -151.8788,B 24.9571,C -1.5128,E1 24.8638,E2 238.0962} C_DIS
LIN {X -103.5821,Y -60.9506,Z 132,A -153.5632,B 24.9571,C -1.5143,E1 24.8614,E2 239.7859} C_DIS
LIN {X -105.5138,Y -57.5404,Z 132,A -155.5686,B 24.9571,C -1.5136,E1 24.8587,E2 241.8036} C_DIS
LIN {X -107.7965,Y -53.1415,Z 132,A -157.8852,B 24.9566,C -1.5222,E1 24.8558,E2 244.112} C_DIS
LIN {X -109.4517,Y -49.6413,Z 132,A -159.6278,B 24.956,C -1.5319,E1 24.8537,E2 245.841} C_DIS
LIN {X -110.8926,Y -46.3348,Z 132,A -161.4658,B 24.956,C -1.5319,E1 24.8517,E2 247.6892} C_DIS
LIN {X -112.3026,Y -42.8039,Z 132,A -163.1815,B 24.9555,C -1.5414,E1 24.85,E2 249.3918} C_DIS
LIN {X -114.2561,Y -37.2764,Z 132,A -166.1599,B 24.9555,C -1.5421,E1 24.8473,E2 252.3856} C_DIS
LIN {X -115.5415,Y -33.079,Z 132,A -168.1978,B 24.9549,C -1.5508,E1 24.8456,E2 254.4145} C_DIS
LIN {X -116.6107,Y -29.0836,Z 132,A -170.074,B 24.9543,C -1.561,E1 24.8443,E2 256.2774} C_DIS
LIN {X -117.5276,Y -25.1301,Z 132,A -172.182,B 24.9544,C -1.5597,E1 24.843,E2 258.4007} C_DIS
LIN {X -118.3154,Y -21.1092,Z 132,A -174.0647,B 24.9539,C -1.5689,E1 24.8421,E2 260.2726} C_DIS
LIN {X -118.9512,Y -17.166,Z 132,A -175.9847,B 24.9536,C -1.5743,E1 24.8413,E2 262.1912} C_DIS
LIN {X -119.3659,Y -13.992,Z 132,A -177.3064,B 24.9528,C -1.5879,E1 24.8408,E2 263.4885} C_DIS
LIN {X -119.6863,Y -10.9207,Z 132,A -178.9918,B 24.953,C -1.5836,E1 24.8403,E2 265.1941} C_DIS
LIN {X -120.002,Y -6.6093,Z 132,A 178.9061,B 24.9527,C -1.5886,E1 24.84,E2 267.297} C_DIS
LIN {X -120.1537,Y -2.6716,Z 132,A 176.9463,B 24.9526,C -1.5913,E1 24.8398,E2 269.2622} C_DIS
LIN {X -120.171,Y 1.7284,Z 132,A 175.1969,B 24.9513,C -1.6128,E1 24.8398,E2 270.9707} C_DIS
LIN {X -120.0891,Y 4.7545,Z 132,A 173.5626,B 24.9515,C -1.6095,E1 24.84,E2 272.6229} C_DIS
LIN {X -119.9069,Y 8.1476,Z 132,A 171.8428,B 24.9514,C -1.6106,E1 24.8402,E2 274.3503} C_DIS
LIN {X -119.4277,Y 13.457,Z 132,A 169.2919,B 24.9509,C -1.6185,E1 24.8409,E2 276.8977} C_DIS
LIN {X -118.8686,Y 17.7333,Z 132,A 167.2245,B 24.9505,C -1.6248,E1 24.8417,E2 278.9625} C_DIS
LIN {X -118.2465,Y 21.4901,Z 132,A 165.3719,B 24.9503,C -1.6291,E1 24.8426,E2 280.8157} C_DIS
LIN {X -117.4191,Y 25.6283,Z 132,A 163.2993,B 24.95,C -1.6331,E1 24.8438,E2 282.8911} C_DIS
LIN {X -116.4137,Y 29.8651,Z 132,A 161.191,B 24.9497,C -1.6385,E1 24.8452,E2 284.9989} C_DIS
LIN {X -115.3529,Y 33.73,Z 132,A 159.4036,B 24.949,C -1.6497,E1 24.8466,E2 286.7698} C_DIS
LIN {X -113.0406,Y 40.8132,Z 132,A 155.8252,B 24.9484,C -1.6599,E1 24.8497,E2 290.3445} C_DIS
LIN {X -111.0963,Y 45.8441,Z 132,A 153.2168,B 24.948,C -1.6663,E1 24.8524,E2 292.9522} C_DIS
LIN {X -109.6684,Y 49.1601,Z 132,A 151.4817,B 24.9477,C -1.671,E1 24.8543,E2 294.6856} C_DIS
LIN {X -107.9588,Y 52.81,Z 132,A 149.6233,B 24.9471,C -1.6795,E1 24.8565,E2 296.5339} C_DIS
LIN {X -105.8175,Y 56.9804,Z 132,A 147.2374,B 24.9471,C -1.6798,E1 24.8596,E2 298.9318} C_DIS
LIN {X -103.8286,Y 60.5282,Z 132,A 145.2517,B 24.9469,C -1.6835,E1 24.8624,E2 300.9189} C_DIS
LIN {X -101.7581,Y 63.9489,Z 132,A 143.3801,B 24.9464,C -1.6905,E1 24.8651,E2 302.7836} C_DIS
LIN {X -98.2134,Y 69.27,Z 132,A 140.2695,B 24.9461,C -1.6964,E1 24.87,E2 305.8954} C_DIS
LIN {X -95.7487,Y 72.6378,Z 132,A 138.2662,B 24.9458,C -1.7013,E1 24.8733,E2 307.8967} C_DIS
LIN {X -93.2602,Y 75.8065,Z 132,A 136.377,B 24.9453,C -1.7078,E1 24.8766,E2 309.7793} C_DIS
LIN {X -90.6604,Y 78.8984,Z 132,A 134.3781,B 24.9453,C -1.7097,E1 24.8803,E2 311.7828} C_DIS
LIN {X -87.8026,Y 82.0662,Z 132,A 132.3953,B 24.9447,C -1.7171,E1 24.884,E2 313.7568} C_DIS
LIN {X -84.9864,Y 84.9785,Z 132,A 130.4237,B 24.9445,C -1.7202,E1 24.8879,E2 315.7295} C_DIS
LIN {X -81.9883,Y 87.875,Z 132,A 128.4547,B 24.9442,C -1.7257,E1 24.8918,E2 317.6935} C_DIS
LIN {X -78.8294,Y 90.7199,Z 132,A 126.3901,B 24.944,C -1.7288,E1 24.8961,E2 319.7589} C_DIS
LIN {X -75.5009,Y 93.5088,Z 132,A 124.2895,B 24.9438,C -1.7321,E1 24.9007,E2 321.8596} C_DIS
LIN {X -72.1415,Y 96.1241,Z 132,A 122.2706,B 24.9435,C -1.7369,E1 24.9051,E2 323.8744} C_DIS
LIN {X -68.7649,Y 98.5671,Z 132,A 120.3379,B 24.943,C -1.7433,E1 24.9095,E2 325.7985} C_DIS
LIN {X -64.2342,Y 101.5776,Z 132,A 116.8669,B 24.9451,C -1.7108,E1 24.9179,E2 329.358} C_DIS
LIN {X -59.2035,Y 104.5905,Z 132,A 114.6516,B 24.9432,C -1.7406,E1 24.9231,E2 331.5089} C_DIS
LIN {X -54.6299,Y 107.0494,Z 132,A 112.4353,B 24.9422,C -1.7561,E1 24.9285,E2 333.6947} C_DIS
LIN {X -51.2373,Y 108.7145,Z 132,A 110.5583,B 24.9422,C -1.7556,E1 24.9332,E2 335.5775} C_DIS
LIN {X -47.6355,Y 110.3393,Z 132,A 108.8378,B 24.9416,C -1.7656,E1 24.9376,E2 337.2783} C_DIS
LIN {X -44.4016,Y 111.681,Z 132,A 107.0383,B 24.9418,C -1.7623,E1 24.9423,E2 339.0899} C_DIS
LIN {X -40.2303,Y 113.2506,Z 132,A 104.8509,B 24.9418,C -1.7623,E1 24.948,E2 341.2817} C_DIS
LIN {X -35.8981,Y 114.698,Z 132,A 102.6243,B 24.9418,C -1.7627,E1 24.9539,E2 343.5113} C_DIS
LIN {X -32.1366,Y 115.8071,Z 132,A 100.8542,B 24.9413,C -1.7692,E1 24.9587,E2 345.2689} C_DIS
LIN {X -28.6332,Y 116.722,Z 132,A 99.2592,B 24.9408,C -1.7767,E1 24.9629,E2 346.8483} C_DIS
LIN {X -25.3714,Y 117.4754,Z 132,A 97.4423,B 24.9414,C -1.7683,E1 24.9679,E2 348.6874} C_DIS
LIN {X -21.2358,Y 118.2925,Z 132,A 95.4859,B 24.9411,C -1.7723,E1 24.9733,E2 350.6364} C_DIS
LIN {X -17.0968,Y 118.9609,Z 132,A 93.4699,B 24.9411,C -1.7729,E1 24.9789,E2 352.6527} C_DIS
LIN {X -12.8482,Y 119.4945,Z 132,A 91.1483,B 24.9418,C -1.7616,E1 24.9854,E2 355.0026} C_DIS
LIN {X -9.4287,Y 119.8129,Z 132,A 89.7919,B 24.941,C -1.7749,E1 24.9891,E2 356.3282} C_DIS
LIN {X -5.3416,Y 120.0651,Z 132,A 87.8868,B 24.9408,C -1.7777,E1 24.9944,E2 358.2271} C_DIS
LIN {X -0.3919,Y 120.1828,Z 132,A 85.546,B 24.9407,C -1.7792,E1 25.0009,E2 360.5645} C_DIS
LIN {X 2.2216,Y 120.1636,Z 132,A 84.0571,B 24.9414,C -1.7684,E1 25.0051,E2 362.0788} C_DIS
LIN {X 6.9558,Y 119.9821,Z 132,A 82.0269,B 24.9407,C -1.7788,E1 25.0107,E2 364.0837} C_DIS
LIN {X 9.8597,Y 119.7776,Z 132,A 80.6546,B 24.9407,C -1.7794,E1 25.0145,E2 365.4538} C_DIS
LIN {X 13.5424,Y 119.4181,Z 132,A 78.9188,B 24.9406,C -1.7804,E1 25.0193,E2 367.186} C_DIS
LIN {X 17.3057,Y 118.9309,Z 132,A 77.0018,B 24.9409,C -1.7751,E1 25.0247,E2 369.1141} C_DIS
LIN {X 21.6345,Y 118.2203,Z 132,A 74.818,B 24.9413,C -1.7701,E1 25.0307,E2 371.3074} C_DIS
LIN {X 26.012,Y 117.3349,Z 132,A 72.8177,B 24.941,C -1.775,E1 25.0361,E2 373.2937} C_DIS
LIN {X 30.0575,Y 116.364,Z 132,A 70.8001,B 24.9411,C -1.7722,E1 25.0416,E2 375.3148} C_DIS
LIN {X 33.7826,Y 115.3377,Z 132,A 68.9311,B 24.9413,C -1.7697,E1 25.0466,E2 377.1867} C_DIS
LIN {X 38.178,Y 113.9587,Z 132,A 66.7796,B 24.9413,C -1.7699,E1 25.0523,E2 379.3335} C_DIS
LIN {X 41.1234,Y 112.9279,Z 132,A 65.2705,B 24.9414,C -1.7676,E1 25.0563,E2 380.8451} C_DIS
LIN {X 44.9337,Y 111.4678,Z 132,A 63.38,B 24.9414,C -1.7681,E1 25.0612,E2 382.73} C_DIS
LIN {X 48.5503,Y 109.9408,Z 132,A 61.4395,B 24.9418,C -1.7628,E1 25.0662,E2 384.6784} C_DIS
LIN {X 52.8204,Y 107.9537,Z 132,A 59.2561,B 24.9418,C -1.763,E1 25.0717,E2 386.8559} C_DIS
LIN {X 56.6468,Y 105.9961,Z 132,A 57.3239,B 24.9416,C -1.7657,E1 25.0764,E2 388.7762} C_DIS
LIN {X 60.4615,Y 103.8676,Z 132,A 55.1877,B 24.9419,C -1.7602,E1 25.0816,E2 390.9191} C_DIS
LIN {X 63.815,Y 101.8426,Z 132,A 53.2585,B 24.9423,C -1.7544,E1 25.0863,E2 392.8559} C_DIS
LIN {X 67.6166,Y 99.3587,Z 132,A 51.0845,B 24.9426,C -1.7504,E1 25.0913,E2 395.032} C_DIS
LIN {X 71.2856,Y 96.7604,Z 132,A 49.0862,B 24.9424,C -1.7535,E1 25.0958,E2 397.016} C_DIS
LIN {X 74.8296,Y 94.0463,Z 132,A 46.8654,B 24.9429,C -1.7452,E1 25.1007,E2 399.2483} C_DIS
LIN {X 78.1852,Y 91.2759,Z 132,A 44.7969,B 24.9432,C -1.7414,E1 25.1052,E2 401.3178} C_DIS
LIN {X 81.2468,Y 88.5613,Z 132,A 42.7575,B 24.9437,C -1.7332,E1 25.1094,E2 403.3683} C_DIS
LIN {X 84.0383,Y 85.9166,Z 132,A 41.0423,B 24.9436,C -1.7349,E1 25.1128,E2 405.0723} C_DIS
LIN {X 87.0158,Y 82.8996,Z 132,A 39.0613,B 24.9438,C -1.7324,E1 25.1167,E2 407.0508} C_DIS
LIN {X 89.7235,Y 79.9613,Z 132,A 37.171,B 24.944,C -1.7287,E1 25.1202,E2 408.9414} C_DIS
LIN {X 93.1742,Y 75.9119,Z 132,A 34.6068,B 24.9445,C -1.7213,E1 25.1248,E2 411.5113} C_DIS
LIN {X 95.7056,Y 72.6948,Z 132,A 32.6451,B 24.9448,C -1.716,E1 25.1282,E2 413.4761} C_DIS
LIN {X 98.0378,Y 69.518,Z 132,A 30.5042,B 24.9459,C -1.6987,E1 25.1317,E2 415.6476} C_DIS
LIN {X 99.9665,Y 66.7145,Z 132,A 29.1705,B 24.9453,C -1.7083,E1 25.1338,E2 416.952} C_DIS
LIN {X 102.0339,Y 63.507,Z 132,A 27.638,B 24.9447,C -1.7174,E1 25.136,E2 418.4554} C_DIS
LIN {X 104.127,Y 60.0147,Z 132,A 25.4538,B 24.9458,C -1.7003,E1 25.1392,E2 420.6686} C_DIS
LIN {X 106.0661,Y 56.516,Z 132,A 23.5453,B 24.9462,C -1.6949,E1 25.1417,E2 422.5799} C_DIS
LIN {X 107.4416,Y 53.8547,Z 132,A 21.7066,B 24.9477,C -1.6711,E1 25.1441,E2 424.465} C_DIS
LIN {X 109.2048,Y 50.185,Z 132,A 20.1497,B 24.9469,C -1.684,E1 25.1459,E2 425.983} C_DIS
LIN {X 110.9565,Y 46.183,Z 132,A 17.7965,B 24.9481,C -1.6648,E1 25.1485,E2 428.3686} C_DIS
LIN {X 112.2755,Y 42.875,Z 132,A 16.4458,B 24.9473,C -1.6766,E1 25.1498,E2 429.684} C_DIS
LIN {X 113.5558,Y 39.3594,Z 132,A 14.652,B 24.9477,C -1.6707,E1 25.1515,E2 431.4816} C_DIS
LIN {X 114.8611,Y 35.369,Z 132,A 12.7193,B 24.9479,C -1.6679,E1 25.1531,E2 433.4098} C_DIS
LIN {X 115.9253,Y 31.7112,Z 132,A 10.8835,B 24.9483,C -1.6613,E1 25.1545,E2 435.2507} C_DIS
LIN {X 116.801,Y 28.309,Z 132,A 9.3571,B 24.9482,C -1.6634,E1 25.1555,E2 436.7634} C_DIS
LIN {X 117.8361,Y 23.6366,Z 132,A 6.9394,B 24.949,C -1.6495,E1 25.1569,E2 439.1998} C_DIS
LIN {X 118.5874,Y 19.523,Z 132,A 5.0358,B 24.9491,C -1.6475,E1 25.1578,E2 441.0968} C_DIS
LIN {X 119.2682,Y 14.8032,Z 132,A 2.6076,B 24.9501,C -1.6326,E1 25.1588,E2 443.5458} C_DIS
LIN {X 119.8154,Y 9.3976,Z 132,A 0.11,B 24.9503,C -1.6288,E1 25.1594,E2 446.0377} C_DIS
LIN {X 120.0254,Y 6.1551,Z 132,A -1.8774,B 24.9519,C -1.6023,E1 25.1597,E2 448.0757} C_DIS
LIN {X 120.1692,Y 1.8578,Z 132,A -3.3535,B 24.9506,C -1.6237,E1 25.1597,E2 449.4928} C_DIS
LIN {X 120.0183,Y -6.2929,Z 132,A -7.0713,B 24.9509,C -1.6192,E1 25.1596,E2 453.1989} C_DIS
LIN {X 119.7882,Y -9.7301,Z 132,A -8.7368,B 24.9513,C -1.6126,E1 25.1592,E2 454.8701} C_DIS
LIN {X 119.4816,Y -12.9725,Z 132,A -10.4101,B 24.9519,C -1.6016,E1 25.1587,E2 456.5595} C_DIS
LIN {X 119.0542,Y -16.4361,Z 132,A -12.0774,B 24.9523,C -1.5959,E1 25.1581,E2 458.2302} C_DIS
LIN {X 118.4655,Y -20.245,Z 132,A -14.1442,B 24.9533,C -1.5787,E1 25.1572,E2 460.3256} C_DIS
LIN {X 117.4971,Y -25.2722,Z 132,A -16.4155,B 24.9533,C -1.579,E1 25.1559,E2 462.5827} C_DIS
LIN {X 116.4682,Y -29.6516,Z 132,A -18.5537,B 24.9537,C -1.5724,E1 25.1545,E2 464.7242} C_DIS
LIN {X 115.4458,Y -33.4093,Z 132,A -20.307,B 24.9537,C -1.5715,E1 25.1532,E2 466.4695} C_DIS
LIN {X 114.3527,Y -36.9775,Z 132,A -22.2317,B 24.9545,C -1.5587,E1 25.1515,E2 468.4135} C_DIS
LIN {X 112.8992,Y -41.2026,Z 132,A -24.1665,B 24.9543,C -1.5616,E1 25.1498,E2 470.3307} C_DIS
LIN {X 111.6926,Y -44.3727,Z 132,A -25.7819,B 24.9546,C -1.5566,E1 25.1481,E2 471.949} C_DIS
LIN {X 110.2262,Y -47.8979,Z 132,A -27.6564,B 24.9551,C -1.5483,E1 25.1461,E2 473.8328} C_DIS
LIN {X 108.6218,Y -51.4328,Z 132,A -29.4888,B 24.9554,C -1.5435,E1 25.1439,E2 475.6666} C_DIS
LIN {X 106.7277,Y -55.2577,Z 132,A -31.5645,B 24.9558,C -1.5353,E1 25.1413,E2 477.7505} C_DIS
LIN {X 104.8364,Y -58.7654,Z 132,A -33.3865,B 24.9559,C -1.5335,E1 25.1388,E2 479.5673} C_DIS
LIN {X 102.7475,Y -62.3459,Z 132,A -35.3401,B 24.9562,C -1.5288,E1 25.136,E2 481.5219} C_DIS
LIN {X 100.5274,Y -65.8668,Z 132,A -37.257,B 24.9564,C -1.5263,E1 25.1332,E2 483.4349} C_DIS
LIN {X 98.6832,Y -68.5981,Z 132,A -38.8934,B 24.9568,C -1.5187,E1 25.1306,E2 485.0813} C_DIS
LIN {X 96.1779,Y -72.0702,Z 132,A -40.9058,B 24.957,C -1.5144,E1 25.1272,E2 487.094} C_DIS
LIN {X 93.9266,Y -74.979,Z 132,A -42.676,B 24.9573,C -1.5089,E1 25.1242,E2 488.869} C_DIS
LIN {X 91.3054,Y -78.151,Z 132,A -44.609,B 24.9576,C -1.5051,E1 25.1207,E2 490.8022} C_DIS
LIN {X 89.1907,Y -80.5555,Z 132,A -46.1926,B 24.9579,C -1.4983,E1 25.1177,E2 492.3946} C_DIS
LIN {X 86.1141,Y -83.8365,Z 132,A -48.2787,B 24.9581,C -1.4957,E1 25.1137,E2 494.4778} C_DIS
LIN {X 83.2169,Y -86.7124,Z 132,A -50.2028,B 24.9583,C -1.492,E1 25.1099,E2 496.4026} C_DIS
LIN {X 80.689,Y -89.0702,Z 132,A -51.8791,B 24.9586,C -1.4867,E1 25.1064,E2 498.0846} C_DIS
LIN {X 77.5849,Y -91.7858,Z 132,A -53.7643,B 24.9586,C -1.4861,E1 25.1024,E2 499.964} C_DIS
LIN {X 74.4855,Y -94.3188,Z 132,A -55.7184,B 24.959,C -1.4796,E1 25.0982,E2 501.926} C_DIS
LIN {X 71.8839,Y -96.3164,Z 132,A -57.2882,B 24.9592,C -1.476,E1 25.0947,E2 503.4987} C_DIS
LIN {X 68.4899,Y -98.7584,Z 132,A -59.1566,B 24.9591,C -1.4778,E1 25.0904,E2 505.3563} C_DIS
LIN {X 65.3975,Y -100.8327,Z 132,A -60.9811,B 24.9594,C -1.4719,E1 25.0861,E2 507.1887} C_DIS
LIN {X 62.3044,Y -102.7727,Z 132,A -62.6358,B 24.9594,C -1.4727,E1 25.0822,E2 508.8364} C_DIS
LIN {X 59.0752,Y -104.6626,Z 132,A -64.5096,B 24.9598,C -1.4651,E1 25.0777,E2 510.7224} C_DIS
LIN {X 55.1485,Y -106.7842,Z 132,A -66.4162,B 24.9594,C -1.472,E1 25.073,E2 512.6074} C_DIS
LIN {X 51.4234,Y -108.6263,Z 132,A -68.5554,B 24.96,C -1.4612,E1 25.0676,E2 514.7664} C_DIS
LIN {X 47.9065,Y -110.2225,Z 132,A -70.4566,B 24.9603,C -1.4555,E1 25.0627,E2 516.6765} C_DIS
LIN {X 44.0684,Y -111.8129,Z 132,A -72.7038,B 24.9612,C -1.44,E1 25.0568,E2 518.9552} C_DIS
LIN {X 40.9943,Y -112.9748,Z 132,A -73.8839,B 24.9603,C -1.4562,E1 25.0538,E2 520.0944} C_DIS
LIN {X 37.4757,Y -114.1907,Z 132,A -75.7396,B 24.9606,C -1.4501,E1 25.0489,E2 521.9609} C_DIS
LIN {X 33.5704,Y -115.3991,Z 132,A -77.7405,B 24.9609,C -1.4454,E1 25.0435,E2 523.9695} C_DIS
LIN {X 29.3328,Y -116.5482,Z 132,A -79.7839,B 24.9609,C -1.4455,E1 25.038,E2 526.0095} C_DIS
LIN {X 25.0744,Y -117.5393,Z 132,A -82.0021,B 24.9613,C -1.4373,E1 25.0319,E2 528.2442} C_DIS
LIN {X 20.4643,Y -118.4282,Z 132,A -83.8349,B 24.9604,C -1.4544,E1 25.027,E2 530.0342} C_DIS
LIN {X 16.1127,Y -119.0985,Z 132,A -86.1834,B 24.9611,C -1.4412,E1 25.0205,E2 532.4119} C_DIS
LIN {X 12.2571,Y -119.5574,Z 132,A -88.559,B 24.9624,C -1.4159,E1 25.0137,E2 534.8459} C_DIS
LIN {X 7.8838,Y -119.9241,Z 132,A -89.8713,B 24.9606,C -1.451,E1 25.0103,E2 536.0744} C_DIS
LIN {X 5.0726,Y -120.0761,Z 132,A -91.9219,B 24.9623,C -1.4177,E1 25.0043,E2 538.2032} C_DIS
LIN {X 0.8571,Y -120.1803,Z 132,A -93.1144,B 24.9603,C -1.4549,E1 25.0013,E2 539.3075} C_DIS
Enddeposition()
LIN {X 0.8571,Y -120.1803,Z 132,A -93.1144,B 24.9603,C -1.4549,E1 25.0013,E2 539.3075} C_DIS
Startdeposition()
$VEL.CP = VEL_PRINT
LIN {X 2.9042,Y -119.31,Z 132,A -91.6676,B 24.9583,C -1.4914,E1 25.0055,E2 537.7744} C_DIS
LIN {X 6.6514,Y -119.1605,Z 132,A -89.8503,B 24.9583,C -1.4929,E1 25.0106,E2 535.9543} C_DIS
LIN {X 9.9251,Y -118.9312,Z 132,A -88.3528,B 24.9584,C -1.49,E1 25.0147,E2 534.4643} C_DIS
LIN {X 13.153,Y -118.6183,Z 132,A -86.7395,B 24.9582,C -1.4935,E1 25.0192,E2 532.8437} C_DIS
LIN {X 16.9697,Y -118.1324,Z 132,A -84.8919,B 24.9582,C -1.4948,E1 25.0244,E2 530.9947} C_DIS
LIN {X 20.3373,Y -117.5997,Z 132,A -83.3667,B 24.9584,C -1.4908,E1 25.0285,E2 529.4806} C_DIS
LIN {X 23.2711,Y -117.0545,Z 132,A -81.8285,B 24.958,C -1.497,E1 25.0328,E2 527.9295} C_DIS
LIN {X 27.0588,Y -116.2375,Z 132,A -79.9453,B 24.9579,C -1.4998,E1 25.0379,E2 526.0421} C_DIS
LIN {X 31.1229,Y -115.2158,Z 132,A -78.0279,B 24.9579,C -1.4975,E1 25.0431,E2 524.1332} C_DIS
LIN {X 34.5759,Y -114.2261,Z 132,A -76.3327,B 24.9579,C -1.4981,E1 25.0476,E2 522.4395} C_DIS
LIN {X 38.3217,Y -113.0254,Z 132,A -74.4979,B 24.9579,C -1.4978,E1 25.0525,E2 520.6088} C_DIS
LIN {X 40.6941,Y -112.1921,Z 132,A -73.2164,B 24.9577,C -1.503,E1 25.0559,E2 519.3176} C_DIS
LIN {X 44.3212,Y -110.8103,Z 132,A -71.2882,B 24.9574,C -1.5087,E1 25.0609,E2 517.3803} C_DIS
LIN {X 47.8751,Y -109.322,Z 132,A -69.452,B 24.9572,C -1.5108,E1 25.0656,E2 515.5434} C_DIS
LIN {X 51.0116,Y -107.8939,Z 132,A -67.8128,B 24.9572,C -1.5127,E1 25.0698,E2 513.9039} C_DIS
LIN {X 54.4567,Y -106.1968,Z 132,A -66.0182,B 24.9571,C -1.5135,E1 25.0743,E2 512.1124} C_DIS
LIN {X 57.7432,Y -104.4474,Z 132,A -64.1329,B 24.9566,C -1.5213,E1 25.0789,E2 510.214} C_DIS
LIN {X 61.3602,Y -102.3635,Z 132,A -62.1775,B 24.9566,C -1.5227,E1 25.0836,E2 508.2612} C_DIS
LIN {X 64.639,Y -100.325,Z 132,A -60.4534,B 24.9567,C -1.5201,E1 25.0876,E2 506.5489} C_DIS
LIN {X 67.5134,Y -98.4135,Z 132,A -58.698,B 24.9562,C -1.5282,E1 25.0917,E2 504.7804} C_DIS
LIN {X 70.6584,Y -96.1813,Z 132,A -56.937,B 24.9562,C -1.5277,E1 25.0957,E2 503.0267} C_DIS
LIN {X 73.0564,Y -94.3721,Z 132,A -55.4195,B 24.9559,C -1.5345,E1 25.0991,E2 501.4986} C_DIS
LIN {X 76.0695,Y -91.9609,Z 132,A -53.5857,B 24.9557,C -1.5377,E1 25.1031,E2 499.6642} C_DIS
LIN {X 79.0467,Y -89.4144,Z 132,A -51.7046,B 24.9554,C -1.5421,E1 25.107,E2 497.7801} C_DIS
LIN {X 81.7636,Y -86.9374,Z 132,A -49.898,B 24.9551,C -1.5484,E1 25.1108,E2 495.9661} C_DIS
LIN {X 84.9017,Y -83.8754,Z 132,A -47.897,B 24.9551,C -1.5484,E1 25.1147,E2 493.9732} C_DIS
LIN {X 87.4293,Y -81.2366,Z 132,A -46.1234,B 24.9548,C -1.5539,E1 25.1181,E2 492.1947} C_DIS
LIN {X 89.891,Y -78.505,Z 132,A -44.385,B 24.9546,C -1.5572,E1 25.1213,E2 490.4563} C_DIS
LIN {X 92.2528,Y -75.7154,Z 132,A -42.6191,B 24.9543,C -1.5624,E1 25.1245,E2 488.6862} C_DIS
LIN {X 94.7601,Y -72.5529,Z 132,A -40.6491,B 24.9539,C -1.5693,E1 25.1279,E2 486.7093} C_DIS
LIN {X 97.271,Y -69.1498,Z 132,A -38.7706,B 24.9539,C -1.5674,E1 25.1309,E2 484.8441} C_DIS
LIN {X 99.2297,Y -66.3089,Z 132,A -36.9997,B 24.9534,C -1.5778,E1 25.1337,E2 483.0576} C_DIS
LIN {X 101.3207,Y -63.0666,Z 132,A -35.2098,B 24.9532,C -1.5801,E1 25.1364,E2 481.2713} C_DIS
LIN {X 103.3754,Y -59.6404,Z 132,A -33.2673,B 24.9528,C -1.5869,E1 25.1392,E2 479.3227} C_DIS
LIN {X 105.0136,Y -56.7062,Z 132,A -31.6532,B 24.9525,C -1.5917,E1 25.1413,E2 477.7056} C_DIS
LIN {X 107.023,Y -52.8152,Z 132,A -29.6507,B 24.9525,C -1.5932,E1 25.1439,E2 475.7104} C_DIS
LIN {X 108.5036,Y -49.7024,Z 132,A -28.0282,B 24.9522,C -1.5966,E1 25.1458,E2 474.0884} C_DIS
LIN {X 109.6876,Y -47.029,Z 132,A -26.5505,B 24.9518,C -1.6047,E1 25.1474,E2 472.5999} C_DIS
LIN {X 111.148,Y -43.4672,Z 132,A -24.8087,B 24.9518,C -1.6052,E1 25.1492,E2 470.8666} C_DIS
LIN {X 112.3683,Y -40.2075,Z 132,A -23.0363,B 24.9511,C -1.6155,E1 25.1509,E2 469.0799} C_DIS
LIN {X 113.6151,Y -36.5334,Z 132,A -21.3266,B 24.9511,C -1.6138,E1 25.1524,E2 467.3837} C_DIS
LIN {X 114.4772,Y -33.7396,Z 132,A -19.7816,B 24.9505,C -1.6253,E1 25.1537,E2 465.8205} C_DIS
LIN {X 115.553,Y -29.8459,Z 132,A -17.7928,B 24.95,C -1.634,E1 25.1551,E2 463.8225} C_DIS
LIN {X 116.4714,Y -26.0319,Z 132,A -16.0051,B 24.9499,C -1.6354,E1 25.1562,E2 462.042} C_DIS
LIN {X 117.2297,Y -22.3696,Z 132,A -14.3499,B 24.9499,C -1.6343,E1 25.1571,E2 460.399} C_DIS
LIN {X 117.8301,Y -18.9569,Z 132,A -12.5554,B 24.9492,C -1.6462,E1 25.158,E2 458.587} C_DIS
LIN {X 118.3807,Y -15.145,Z 132,A -10.7155,B 24.9489,C -1.6518,E1 25.1587,E2 456.7447} C_DIS
LIN {X 118.7684,Y -11.7191,Z 132,A -9.0655,B 24.9486,C -1.657,E1 25.1592,E2 455.0923} C_DIS
LIN {X 119.0836,Y -7.894,Z 132,A -7.248,B 24.9483,C -1.6618,E1 25.1595,E2 453.2743} C_DIS
LIN {X 119.2808,Y -3.9164,Z 132,A -5.4146,B 24.9481,C -1.6641,E1 25.1597,E2 451.4462} C_DIS
LIN {X 119.3458,Y -0.1339,Z 132,A -3.6168,B 24.9478,C -1.6692,E1 25.1597,E2 449.6471} C_DIS
LIN {X 119.31,Y 2.9017,Z 132,A -2.1055,B 24.9473,C -1.6766,E1 25.1597,E2 448.1273} C_DIS
LIN {X 119.1522,Y 6.7924,Z 132,A -0.2488,B 24.947,C -1.6821,E1 25.1594,E2 446.2688} C_DIS
LIN {X 118.9068,Y 10.2212,Z 132,A 1.3767,B 24.9467,C -1.6862,E1 25.1591,E2 444.6432} C_DIS
LIN {X 118.5179,Y 14.0283,Z 132,A 3.2181,B 24.9463,C -1.6924,E1 25.1585,E2 442.7982} C_DIS
LIN {X 117.9746,Y 18.0353,Z 132,A 5.124,B 24.946,C -1.6969,E1 25.1578,E2 440.8929} C_DIS
LIN {X 117.3314,Y 21.8342,Z 132,A 6.8858,B 24.946,C -1.6984,E1 25.1569,E2 439.1379} C_DIS
LIN {X 116.7621,Y 24.6969,Z 132,A 8.2824,B 24.9457,C -1.7026,E1 25.1561,E2 437.7394} C_DIS
LIN {X 116.1238,Y 27.5422,Z 132,A 9.7702,B 24.9451,C -1.7113,E1 25.1552,E2 436.2397} C_DIS
LIN {X 115.0229,Y 31.8282,Z 132,A 11.8679,B 24.9448,C -1.7166,E1 25.1537,E2 434.1416} C_DIS
LIN {X 113.9133,Y 35.5991,Z 132,A 13.8234,B 24.9442,C -1.7258,E1 25.1521,E2 432.1756} C_DIS
LIN {X 112.5456,Y 39.7112,Z 132,A 15.8362,B 24.944,C -1.7288,E1 25.1502,E2 430.1671} C_DIS
LIN {X 111.0123,Y 43.8142,Z 132,A 17.9224,B 24.9436,C -1.7342,E1 25.1482,E2 428.0797} C_DIS
LIN {X 109.4023,Y 47.6908,Z 132,A 19.7842,B 24.9437,C -1.7326,E1 25.1461,E2 426.2319} C_DIS
LIN {X 108.1201,Y 50.5304,Z 132,A 21.4019,B 24.9431,C -1.7429,E1 25.1442,E2 424.5987} C_DIS
LIN {X 106.2092,Y 54.4324,Z 132,A 23.4896,B 24.9427,C -1.7489,E1 25.1416,E2 422.5079} C_DIS
LIN {X 104.3007,Y 58.006,Z 132,A 25.3669,B 24.9425,C -1.751,E1 25.1391,E2 420.6356} C_DIS
LIN {X 102.3717,Y 61.3466,Z 132,A 27.2604,B 24.9421,C -1.7581,E1 25.1364,E2 418.7351} C_DIS
LIN {X 100.3269,Y 64.636,Z 132,A 28.9453,B 24.9423,C -1.7545,E1 25.1339,E2 417.0671} C_DIS
LIN {X 98.4209,Y 67.5026,Z 132,A 30.7289,B 24.9416,C -1.7652,E1 25.1311,E2 415.2672} C_DIS
LIN {X 96.2866,Y 70.514,Z 132,A 32.5468,B 24.9412,C -1.7719,E1 25.1281,E2 413.4423} C_DIS
LIN {X 93.636,Y 73.9979,Z 132,A 34.5836,B 24.941,C -1.7739,E1 25.1247,E2 411.4103} C_DIS
LIN {X 91.19,Y 76.9915,Z 132,A 36.4296,B 24.9408,C -1.7779,E1 25.1214,E2 409.5634} C_DIS
LIN {X 88.4317,Y 80.1452,Z 132,A 38.488,B 24.9403,C -1.7848,E1 25.1175,E2 407.4979} C_DIS
LIN {X 85.6104,Y 83.1518,Z 132,A 40.4139,B 24.9402,C -1.7866,E1 25.1138,E2 405.576} C_DIS
LIN {X 82.7918,Y 85.9581,Z 132,A 42.3507,B 24.9398,C -1.792,E1 25.1099,E2 403.6345} C_DIS
LIN {X 80.1449,Y 88.432,Z 132,A 44.089,B 24.9396,C -1.7955,E1 25.1064,E2 401.8949} C_DIS
LIN {X 77.1973,Y 91.0157,Z 132,A 45.8938,B 24.9396,C -1.7955,E1 25.1026,E2 400.0971} C_DIS
LIN {X 74.003,Y 93.6319,Z 132,A 47.9395,B 24.9391,C -1.8024,E1 25.0981,E2 398.0431} C_DIS
LIN {X 70.8623,Y 96.0308,Z 132,A 49.8139,B 24.939,C -1.8047,E1 25.0939,E2 396.1699} C_DIS
LIN {X 67.9571,Y 98.108,Z 132,A 51.4858,B 24.9389,C -1.8056,E1 25.0901,E2 394.5017} C_DIS
LIN {X 65.0783,Y 100.0409,Z 132,A 53.0499,B 24.939,C -1.8036,E1 25.0865,E2 392.9476} C_DIS
LIN {X 62.1637,Y 101.8773,Z 132,A 54.7552,B 24.9387,C -1.8086,E1 25.0824,E2 391.2359} C_DIS
LIN {X 58.8408,Y 103.8326,Z 132,A 56.698,B 24.9382,C -1.8156,E1 25.0777,E2 389.2823} C_DIS
LIN {X 54.9646,Y 105.9352,Z 132,A 58.8428,B 24.9379,C -1.8198,E1 25.0724,E2 387.1336} C_DIS
LIN {X 51.5047,Y 107.6588,Z 132,A 60.5869,B 24.9381,C -1.8169,E1 25.068,E2 385.401} C_DIS
LIN {X 48.3624,Y 109.1071,Z 132,A 62.1746,B 24.9382,C -1.8154,E1 25.064,E2 383.8209} C_DIS
LIN {X 45.1935,Y 110.4573,Z 132,A 63.8864,B 24.9379,C -1.8199,E1 25.0596,E2 382.1025} C_DIS
LIN {X 42.0956,Y 111.6742,Z 132,A 65.3902,B 24.9381,C -1.8171,E1 25.0557,E2 380.6085} C_DIS
LIN {X 39.0264,Y 112.7842,Z 132,A 67.0885,B 24.9376,C -1.8246,E1 25.0512,E2 378.8959} C_DIS
LIN {X 35.1435,Y 114.0535,Z 132,A 69.0428,B 24.9376,C -1.8258,E1 25.046,E2 376.9422} C_DIS
LIN {X 31.3233,Y 115.162,Z 132,A 71.052,B 24.9371,C -1.8318,E1 25.0405,E2 374.9222} C_DIS
LIN {X 27.0701,Y 116.2349,Z 132,A 73.0096,B 24.9375,C -1.8261,E1 25.0353,E2 372.9809} C_DIS
LIN {X 24.2136,Y 116.8624,Z 132,A 74.4078,B 24.9375,C -1.8265,E1 25.0315,E2 371.5834} C_DIS
LIN {X 20.9211,Y 117.4977,Z 132,A 76.0613,B 24.9373,C -1.8292,E1 25.0269,E2 369.9256} C_DIS
LIN {X 16.9993,Y 118.1282,Z 132,A 77.9179,B 24.9374,C -1.8274,E1 25.0218,E2 368.0748} C_DIS
LIN {X 13.1704,Y 118.6163,Z 132,A 79.6986,B 24.9376,C -1.8245,E1 25.0169,E2 366.3024} C_DIS
LIN {X 9.7118,Y 118.9487,Z 132,A 81.4422,B 24.9374,C -1.8281,E1 25.012,E2 364.5512} C_DIS
LIN {X 5.8645,Y 119.2011,Z 132,A 83.3324,B 24.9372,C -1.8299,E1 25.0067,E2 362.6577} C_DIS
LIN {X 2.0198,Y 119.3287,Z 132,A 85.0851,B 24.9375,C -1.8254,E1 25.0019,E2 360.9159} C_DIS
LIN {X -1.4495,Y 119.3366,Z 132,A 86.7281,B 24.9376,C -1.824,E1 24.9973,E2 359.2761} C_DIS
LIN {X -4.9144,Y 119.244,Z 132,A 88.466,B 24.9374,C -1.8268,E1 24.9924,E2 357.5313} C_DIS
LIN {X -8.7564,Y 119.0241,Z 132,A 90.2548,B 24.9377,C -1.8234,E1 24.9875,E2 355.75} C_DIS
LIN {X -12.1621,Y 118.7246,Z 132,A 91.9922,B 24.9374,C -1.8269,E1 24.9826,E2 354.0033} C_DIS
LIN {X -16.0604,Y 118.2598,Z 132,A 93.8908,B 24.9374,C -1.8264,E1 24.9773,E2 352.1046} C_DIS
LIN {X -20.0056,Y 117.656,Z 132,A 95.7498,B 24.9377,C -1.8225,E1 24.9722,E2 350.2531} C_DIS
LIN {X -23.265,Y 117.0557,Z 132,A 97.393,B 24.9377,C -1.8235,E1 24.9677,E2 348.6057} C_DIS
LIN {X -27.0649,Y 116.236,Z 132,A 99.2912,B 24.9377,C -1.8232,E1 24.9625,E2 346.7058} C_DIS
LIN {X -31.3167,Y 115.1638,Z 132,A 101.4095,B 24.9377,C -1.8217,E1 24.9568,E2 344.588} C_DIS
LIN {X -34.6355,Y 114.208,Z 132,A 102.8974,B 24.9384,C -1.8123,E1 24.9529,E2 343.1199} C_DIS
LIN {X -37.6044,Y 113.2657,Z 132,A 104.5653,B 24.938,C -1.8181,E1 24.9484,E2 341.4351} C_DIS
LIN {X -41.5945,Y 111.8627,Z 132,A 106.5025,B 24.9385,C -1.8114,E1 24.9434,E2 339.5101} C_DIS
LIN {X -44.3217,Y 110.8101,Z 132,A 107.8604,B 24.9388,C -1.8074,E1 24.9398,E2 338.1586} C_DIS
LIN {X -47.8827,Y 109.3187,Z 132,A 109.7562,B 24.9388,C -1.8066,E1 24.935,E2 336.2605} C_DIS
LIN {X -51.0225,Y 107.8887,Z 132,A 111.4941,B 24.9388,C -1.8076,E1 24.9306,E2 334.5158} C_DIS
LIN {X -54.4817,Y 106.184,Z 132,A 113.3652,B 24.9389,C -1.8054,E1 24.9259,E2 332.6449} C_DIS
LIN {X -57.8727,Y 104.3751,Z 132,A 115.2183,B 24.9391,C -1.8025,E1 24.9213,E2 330.7934} C_DIS
LIN {X -61.3336,Y 102.3794,Z 132,A 117.1434,B 24.9393,C -1.7993,E1 24.9167,E2 328.87} C_DIS
LIN {X -64.5593,Y 100.3763,Z 132,A 118.8554,B 24.9399,C -1.791,E1 24.9127,E2 327.1724} C_DIS
LIN {X -67.3675,Y 98.5137,Z 132,A 120.5729,B 24.9399,C -1.7921,E1 24.9087,E2 325.4465} C_DIS
LIN {X -70.6769,Y 96.1677,Z 132,A 122.5679,B 24.9399,C -1.7902,E1 24.9042,E2 323.4493} C_DIS
LIN {X -73.6333,Y 93.9225,Z 132,A 124.3185,B 24.9403,C -1.785,E1 24.9003,E2 321.7046} C_DIS
LIN {X -76.6329,Y 91.4925,Z 132,A 126.2391,B 24.9403,C -1.7837,E1 24.8962,E2 319.7797} C_DIS
LIN {X -79.8677,Y 88.6823,Z 132,A 128.3053,B 24.9407,C -1.7793,E1 24.8919,E2 317.7157} C_DIS
LIN {X -82.8227,Y 85.9283,Z 132,A 130.202,B 24.9411,C -1.7729,E1 24.888,E2 315.8266} C_DIS
LIN {X -85.5994,Y 83.1632,Z 132,A 132.1191,B 24.9413,C -1.7698,E1 24.8843,E2 313.9087} C_DIS
LIN {X -88.4236,Y 80.1541,Z 132,A 134.1527,B 24.9415,C -1.767,E1 24.8804,E2 311.8728} C_DIS
LIN {X -91.016,Y 77.197,Z 132,A 135.9795,B 24.942,C -1.7595,E1 24.8771,E2 310.0557} C_DIS
LIN {X -93.6291,Y 74.0066,Z 132,A 138.0476,B 24.942,C -1.7579,E1 24.8735,E2 307.9815} C_DIS
LIN {X -96.0159,Y 70.8824,Z 132,A 139.9306,B 24.9424,C -1.7526,E1 24.8703,E2 306.1022} C_DIS
LIN {X -98.1339,Y 67.9198,Z 132,A 141.6488,B 24.9428,C -1.7464,E1 24.8676,E2 304.3903} C_DIS
LIN {X -100.3342,Y 64.6247,Z 132,A 143.5436,B 24.9432,C -1.7407,E1 24.8647,E2 302.4996} C_DIS
LIN {X -102.296,Y 61.4731,Z 132,A 145.3841,B 24.9434,C -1.738,E1 24.862,E2 300.656} C_DIS
LIN {X -104.2635,Y 58.0725,Z 132,A 147.132,B 24.9441,C -1.7266,E1 24.8596,E2 298.9262} C_DIS
LIN {X -105.9253,Y 54.9834,Z 132,A 149.0149,B 24.9439,C -1.73,E1 24.8572,E2 297.0252} C_DIS
LIN {X -107.6602,Y 51.5017,Z 132,A 150.8118,B 24.9445,C -1.7214,E1 24.855,E2 295.2391} C_DIS
LIN {X -109.3167,Y 47.8873,Z 132,A 152.8435,B 24.9445,C -1.7207,E1 24.8526,E2 293.1978} C_DIS
LIN {X -111.1079,Y 43.5696,Z 132,A 154.9304,B 24.9454,C -1.7071,E1 24.8505,E2 291.1318} C_DIS
LIN {X -112.3657,Y 40.2147,Z 132,A 156.7416,B 24.9454,C -1.7055,E1 24.8487,E2 289.314} C_DIS
LIN {X -113.5978,Y 36.5871,Z 132,A 158.4483,B 24.9462,C -1.6941,E1 24.8473,E2 287.6249} C_DIS
LIN {X -114.4761,Y 33.7431,Z 132,A 160.0474,B 24.946,C -1.6967,E1 24.846,E2 286.0103} C_DIS
LIN {X -115.6384,Y 29.5148,Z 132,A 162.1101,B 24.9466,C -1.6882,E1 24.8445,E2 283.956} C_DIS
LIN {X -116.4532,Y 26.1122,Z 132,A 163.8526,B 24.9468,C -1.6854,E1 24.8434,E2 282.2098} C_DIS
LIN {X -117.2322,Y 22.3567,Z 132,A 165.5594,B 24.9475,C -1.6737,E1 24.8425,E2 280.5207} C_DIS
LIN {X -117.8298,Y 18.959,Z 132,A 167.3763,B 24.9475,C -1.6751,E1 24.8416,E2 278.6897} C_DIS
LIN {X -118.3815,Y 15.1385,Z 132,A 169.2449,B 24.9478,C -1.6697,E1 24.8409,E2 276.8228} C_DIS
LIN {X -118.7695,Y 11.7077,Z 132,A 170.9264,B 24.948,C -1.6653,E1 24.8404,E2 275.1418} C_DIS
LIN {X -119.0869,Y 7.8429,Z 132,A 172.7694,B 24.9485,C -1.6584,E1 24.8401,E2 273.3041} C_DIS
LIN {X -119.2821,Y 3.8749,Z 132,A 174.6619,B 24.9489,C -1.6516,E1 24.8398,E2 271.4166} C_DIS
LIN {X -119.3464,Y 0.0015,Z 132,A 176.5792,B 24.9491,C -1.6479,E1 24.8398,E2 269.4965} C_DIS
LIN {X -119.2823,Y -3.8699,Z 132,A 178.44,B 24.9495,C -1.6419,E1 24.8399,E2 267.6387} C_DIS
LIN {X -119.0871,Y -7.8397,Z 132,A -179.6484,B 24.9499,C -1.6359,E1 24.8402,E2 265.73} C_DIS
LIN {X -118.7714,Y -11.6879,Z 132,A -177.8854,B 24.9505,C -1.626,E1 24.8407,E2 263.9799} C_DIS
LIN {X -118.3818,Y -15.1361,Z 132,A -176.0994,B 24.9505,C -1.6257,E1 24.8413,E2 262.184} C_DIS
LIN {X -117.8301,Y -18.9566,Z 132,A -174.2364,B 24.9508,C -1.6202,E1 24.842,E2 260.323} C_DIS
LIN {X -117.1181,Y -22.9476,Z 132,A -172.1979,B 24.9509,C -1.618,E1 24.8431,E2 258.2778} C_DIS
LIN {X -116.2362,Y -27.0642,Z 132,A -170.2045,B 24.9514,C -1.6104,E1 24.8443,E2 256.2906} C_DIS
LIN {X -115.1635,Y -31.3178,Z 132,A -168.1992,B 24.9521,C -1.5996,E1 24.8457,E2 254.2995} C_DIS
LIN {X -114.3157,Y -34.281,Z 132,A -166.6608,B 24.9521,C -1.5976,E1 24.8469,E2 252.7571} C_DIS
LIN {X -113.0807,Y -38.1581,Z 132,A -164.7279,B 24.9526,C -1.5907,E1 24.8486,E2 250.8294} C_DIS
LIN {X -111.6788,Y -42.0834,Z 132,A -162.6036,B 24.9526,C -1.59,E1 24.8507,E2 248.6948} C_DIS
LIN {X -110.261,Y -45.6714,Z 132,A -160.6815,B 24.9528,C -1.5875,E1 24.8527,E2 246.7679} C_DIS
LIN {X -108.5087,Y -49.6911,Z 132,A -158.7571,B 24.9536,C -1.5737,E1 24.8548,E2 244.866} C_DIS
LIN {X -107.1329,Y -52.5908,Z 132,A -157.0771,B 24.9536,C -1.5753,E1 24.8569,E2 243.1731} C_DIS
LIN {X -105.492,Y -55.8097,Z 132,A -155.3694,B 24.9539,C -1.5693,E1 24.8591,E2 241.4706} C_DIS
LIN {X -103.8377,Y -58.8319,Z 132,A -153.6949,B 24.9541,C -1.5656,E1 24.8614,E2 239.7961} C_DIS
LIN {X -101.881,Y -62.1575,Z 132,A -151.8294,B 24.9543,C -1.5612,E1 24.8641,E2 237.9314} C_DIS
LIN {X -99.6516,Y -65.6722,Z 132,A -149.9258,B 24.9549,C -1.5518,E1 24.8669,E2 236.0404} C_DIS
LIN {X -97.5033,Y -68.8228,Z 132,A -147.916,B 24.9547,C -1.5549,E1 24.8702,E2 234.0135} C_DIS
LIN {X -94.9781,Y -72.2667,Z 132,A -145.8827,B 24.955,C -1.5491,E1 24.8735,E2 231.9843} C_DIS
LIN {X -92.4311,Y -75.4969,Z 132,A -143.9938,B 24.9555,C -1.5406,E1 24.8768,E2 230.1068} C_DIS
LIN {X -90.0652,Y -78.3052,Z 132,A -142.1986,B 24.9557,C -1.5378,E1 24.8801,E2 228.3098} C_DIS
LIN {X -87.6244,Y -81.0266,Z 132,A -140.4483,B 24.9559,C -1.5337,E1 24.8834,E2 226.5618} C_DIS
LIN {X -84.9114,Y -83.8656,Z 132,A -138.463,B 24.9559,C -1.5339,E1 24.8873,E2 224.5674} C_DIS
LIN {X -81.7846,Y -86.9176,Z 132,A -136.3553,B 24.9561,C -1.5299,E1 24.8915,E2 222.4604} C_DIS
LIN {X -78.5081,Y -89.8883,Z 132,A -134.305,B 24.9566,C -1.5225,E1 24.8958,E2 220.4197} C_DIS
LIN {X -75.7152,Y -92.253,Z 132,A -132.5215,B 24.9566,C -1.5203,E1 24.8996,E2 218.6346} C_DIS
LIN {X -72.639,Y -94.6939,Z 132,A -130.6109,B 24.9568,C -1.5179,E1 24.9038,E2 216.7226} C_DIS
LIN {X -69.9177,Y -96.7208,Z 132,A -129.0807,B 24.9572,C -1.5107,E1 24.9072,E2 215.2042} C_DIS
LIN {X -67.0801,Y -98.7101,Z 132,A -127.3401,B 24.9572,C -1.5113,E1 24.9112,E2 213.4561} C_DIS
LIN {X -63.8543,Y -100.8261,Z 132,A -125.4485,B 24.9572,C -1.5102,E1 24.9157,E2 211.5612} C_DIS
LIN {X -60.5677,Y -102.8349,Z 132,A -123.5859,B 24.9574,C -1.508,E1 24.9202,E2 209.6981} C_DIS
LIN {X -56.9692,Y -104.871,Z 132,A -121.5337,B 24.9574,C -1.5083,E1 24.9252,E2 207.6393} C_DIS
LIN {X -52.8132,Y -107.024,Z 132,A -119.4269,B 24.9579,C -1.4991,E1 24.9304,E2 205.5486} C_DIS
LIN {X -49.7014,Y -108.504,Z 132,A -117.7905,B 24.9581,C -1.4964,E1 24.9345,E2 203.9146} C_DIS
LIN {X -47.0286,Y -109.6878,Z 132,A -116.2989,B 24.9579,C -1.4988,E1 24.9384,E2 202.4138} C_DIS
LIN {X -43.4672,Y -111.148,Z 132,A -114.5271,B 24.9582,C -1.4935,E1 24.9429,E2 200.6506} C_DIS
LIN {X -40.3309,Y -112.324,Z 132,A -112.788,B 24.958,C -1.498,E1 24.9475,E2 198.8974} C_DIS
LIN {X -36.5415,Y -113.6125,Z 132,A -111.0347,B 24.9585,C -1.4888,E1 24.9521,E2 197.1627} C_DIS
LIN {X -33.2411,Y -114.6219,Z 132,A -109.2632,B 24.9583,C -1.4928,E1 24.9569,E2 195.3787} C_DIS
LIN {X -29.0044,Y -115.7665,Z 132,A -107.1461,B 24.9583,C -1.492,E1 24.9626,E2 193.2603} C_DIS
LIN {X -25.2503,Y -116.6439,Z 132,A -105.4169,B 24.9587,C -1.4855,E1 24.9673,E2 191.5443} C_DIS
LIN {X -22.3657,Y -117.2305,Z 132,A -103.9973,B 24.9587,C -1.4852,E1 24.9712,E2 190.1238} C_DIS
LIN {X -18.9696,Y -117.828,Z 132,A -102.1969,B 24.9583,C -1.4914,E1 24.9762,E2 188.3072} C_DIS
LIN {X -15.1611,Y -118.3787,Z 132,A -100.3407,B 24.9583,C -1.4914,E1 24.9813,E2 186.4495} C_DIS
LIN {X -11.6987,Y -118.7704,Z 132,A -98.6629,B 24.9583,C -1.4914,E1 24.986,E2 184.7706} C_DIS
LIN {X -7.8645,Y -119.0855,Z 132,A -96.8395,B 24.9583,C -1.4903,E1 24.9911,E2 182.949} C_DIS
LIN {X -3.8804,Y -119.2819,Z 132,A -94.9661,B 24.9585,C -1.4886,E1 24.9963,E2 181.0794} C_DIS
LIN {X -0.5769,Y -119.3439,Z 132,A -93.4652,B 24.9587,C -1.4849,E1 25.0005,E2 179.5871} C_DIS
LIN {X -0.5769,Y -119.3439,Z 132,A -93.4652,B 24.9587,C -1.4849,E1 25.0005,E2 179.5871} C_DIS
Enddeposition()
LIN {X 0.8871,Y -124.866,Z 133,A -92.6313,B 24.9631,C -1.4037,E1 25.0022,E2 178.9456} C_DIS
Startdeposition()
$VEL.CP = VEL_PRINT
LIN {X -3.4502,Y -124.8224,Z 133,A -95.2436,B 24.9647,C -1.3731,E1 24.9948,E2 181.6307} C_DIS
LIN {X -6.824,Y -124.6859,Z 133,A -96.7477,B 24.9646,C -1.3751,E1 24.9906,E2 183.1303} C_DIS
LIN {X -11.1576,Y -124.3726,Z 133,A -98.8662,B 24.9649,C -1.3692,E1 24.9846,E2 185.2639} C_DIS
LIN {X -14.8682,Y -123.9817,Z 133,A -100.5057,B 24.9647,C -1.3729,E1 24.9801,E2 186.8956} C_DIS
LIN {X -18.2642,Y -123.5297,Z 133,A -102.0275,B 24.9646,C -1.3756,E1 24.9759,E2 188.4121} C_DIS
LIN {X -21.2737,Y -123.0464,Z 133,A -103.3726,B 24.9644,C -1.3786,E1 24.9722,E2 189.7513} C_DIS
LIN {X -23.9077,Y -122.5611,Z 133,A -104.6143,B 24.9644,C -1.3785,E1 24.9688,E2 190.9947} C_DIS
LIN {X -27.0788,Y -121.9008,Z 133,A -106.0908,B 24.9644,C -1.3796,E1 24.9648,E2 192.4703} C_DIS
LIN {X -29.5009,Y -121.3353,Z 133,A -107.3162,B 24.9645,C -1.3763,E1 24.9614,E2 193.7053} C_DIS
LIN {X -32.8189,Y -120.4825,Z 133,A -108.8678,B 24.9645,C -1.3781,E1 24.9572,E2 195.2548} C_DIS
LIN {X -35.8156,Y -119.6254,Z 133,A -110.2467,B 24.9642,C -1.3816,E1 24.9536,E2 196.6278} C_DIS
LIN {X -38.3543,Y -118.8346,Z 133,A -111.5585,B 24.9644,C -1.3782,E1 24.95,E2 197.9499} C_DIS
LIN {X -41.6005,Y -117.7396,Z 133,A -113.0976,B 24.9643,C -1.381,E1 24.946,E2 199.4853} C_DIS
LIN {X -44.4583,Y -116.6895,Z 133,A -114.4644,B 24.9641,C -1.3838,E1 24.9424,E2 200.8484} C_DIS
LIN {X -46.9533,Y -115.7063,Z 133,A -115.771,B 24.9643,C -1.3815,E1 24.939,E2 202.1633} C_DIS
LIN {X -50.1104,Y -114.376,Z 133,A -117.2845,B 24.964,C -1.3859,E1 24.9352,E2 203.6699} C_DIS
LIN {X -53.0574,Y -113.0397,Z 133,A -118.7682,B 24.964,C -1.3877,E1 24.9314,E2 205.153} C_DIS
LIN {X -55.3887,Y -111.9131,Z 133,A -120.0167,B 24.964,C -1.3863,E1 24.9282,E2 206.4079} C_DIS
LIN {X -58.7517,Y -110.1873,Z 133,A -121.7998,B 24.964,C -1.3863,E1 24.9238,E2 208.196} C_DIS
LIN {X -62.2484,Y -108.2507,Z 133,A -123.715,B 24.964,C -1.3851,E1 24.9191,E2 210.1196} C_DIS
LIN {X -66.3133,Y -105.81,Z 133,A -125.7656,B 24.9636,C -1.3942,E1 24.9143,E2 212.155} C_DIS
LIN {X -69.2398,Y -103.9169,Z 133,A -127.435,B 24.9636,C -1.3936,E1 24.9104,E2 213.8313} C_DIS
LIN {X -72.9272,Y -101.3646,Z 133,A -129.4448,B 24.9633,C -1.3993,E1 24.9058,E2 215.8346} C_DIS
LIN {X -75.5403,Y -99.4318,Z 133,A -130.9326,B 24.9632,C -1.4021,E1 24.9025,E2 217.3209} C_DIS
LIN {X -78.7067,Y -96.9448,Z 133,A -132.8794,B 24.9632,C -1.401,E1 24.8982,E2 219.2777} C_DIS
LIN {X -81.7962,Y -94.3527,Z 133,A -134.7747,B 24.9632,C -1.4025,E1 24.8942,E2 221.1766} C_DIS
LIN {X -84.8038,Y -91.6588,Z 133,A -136.5759,B 24.9628,C -1.4087,E1 24.8905,E2 222.9704} C_DIS
LIN {X -87.7247,Y -88.8677,Z 133,A -138.5062,B 24.9628,C -1.4091,E1 24.8866,E2 224.9078} C_DIS
LIN {X -90.5292,Y -86.0086,Z 133,A -140.2765,B 24.9624,C -1.4162,E1 24.8832,E2 226.6688} C_DIS
LIN {X -93.2873,Y -83.0096,Z 133,A -142.2107,B 24.9624,C -1.4175,E1 24.8795,E2 228.6084} C_DIS
LIN {X -95.8935,Y -79.984,Z 133,A -143.9853,B 24.962,C -1.4245,E1 24.8764,E2 230.3747} C_DIS
LIN {X -98.4502,Y -76.816,Z 133,A -145.9478,B 24.962,C -1.4247,E1 24.8729,E2 232.3458} C_DIS
LIN {X -100.8511,Y -73.6345,Z 133,A -147.694,B 24.9615,C -1.433,E1 24.87,E2 234.0806} C_DIS
LIN {X -103.1645,Y -70.3577,Z 133,A -149.6448,B 24.9615,C -1.4328,E1 24.8669,E2 236.0416} C_DIS
LIN {X -105.3831,Y -66.9879,Z 133,A -151.4008,B 24.9611,C -1.4419,E1 24.8643,E2 237.7847} C_DIS
LIN {X -107.4674,Y -63.5914,Z 133,A -153.3392,B 24.9611,C -1.4419,E1 24.8615,E2 239.7331} C_DIS
LIN {X -109.8114,Y -59.4535,Z 133,A -155.5236,B 24.9607,C -1.4478,E1 24.8585,E2 241.915} C_DIS
LIN {X -111.3984,Y -56.4174,Z 133,A -156.9957,B 24.9602,C -1.4568,E1 24.8567,E2 243.3736} C_DIS
LIN {X -112.8616,Y -53.4328,Z 133,A -158.5428,B 24.9601,C -1.4601,E1 24.8548,E2 244.9211} C_DIS
LIN {X -114.3064,Y -50.2713,Z 133,A -160.0884,B 24.9597,C -1.4669,E1 24.853,E2 246.459} C_DIS
LIN {X -115.2685,Y -48.0169,Z 133,A -161.2554,B 24.9597,C -1.4684,E1 24.8518,E2 247.629} C_DIS
LIN {X -116.5256,Y -44.8832,Z 133,A -162.8286,B 24.9594,C -1.4719,E1 24.8502,E2 249.2026} C_DIS
LIN {X -117.7148,Y -41.6703,Z 133,A -164.3716,B 24.9591,C -1.4779,E1 24.8487,E2 250.7401} C_DIS
LIN {X -118.6089,Y -39.0458,Z 133,A -165.6374,B 24.9589,C -1.4821,E1 24.8476,E2 252.0031} C_DIS
LIN {X -119.4994,Y -36.2295,Z 133,A -167.0442,B 24.9587,C -1.4839,E1 24.8464,E2 253.4136} C_DIS
LIN {X -120.4422,Y -32.9677,Z 133,A -168.5783,B 24.9584,C -1.4898,E1 24.8452,E2 254.9426} C_DIS
LIN {X -121.0581,Y -30.6172,Z 133,A -169.7426,B 24.9584,C -1.4911,E1 24.8444,E2 256.1106} C_DIS
LIN {X -121.8429,Y -27.3332,Z 133,A -171.2195,B 24.9579,C -1.4992,E1 24.8435,E2 257.577} C_DIS
LIN {X -122.5102,Y -24.1727,Z 133,A -172.694,B 24.9576,C -1.5042,E1 24.8427,E2 259.0482} C_DIS
LIN {X -122.9671,Y -21.7186,Z 133,A -173.9487,B 24.9576,C -1.503,E1 24.8421,E2 260.3131} C_DIS
LIN {X -123.5964,Y -17.795,Z 133,A -175.7986,B 24.9574,C -1.5077,E1 24.8413,E2 262.1629} C_DIS
LIN {X -124.0763,Y -14.0747,Z 133,A -177.4124,B 24.9568,C -1.5179,E1 24.8407,E2 263.7619} C_DIS
LIN {X -124.3421,Y -11.4861,Z 133,A -178.6512,B 24.9568,C -1.5198,E1 24.8404,E2 265.0036} C_DIS
LIN {X -124.5859,Y -8.4462,Z 133,A 179.9675,B 24.9564,C -1.5252,E1 24.8401,E2 266.3804} C_DIS
LIN {X -124.7483,Y -5.5668,Z 133,A 178.413,B 24.9568,C -1.5193,E1 24.8399,E2 267.9584} C_DIS
LIN {X -124.8637,Y -1.4441,Z 133,A 176.7345,B 24.9559,C -1.5349,E1 24.8398,E2 269.6098} C_DIS
LIN {X -124.8646,Y 1.3828,Z 133,A 175.2055,B 24.9562,C -1.5289,E1 24.8398,E2 271.1622} C_DIS
LIN {X -124.7508,Y 5.505,Z 133,A 173.524,B 24.9553,C -1.5444,E1 24.84,E2 272.8169} C_DIS
LIN {X -124.5347,Y 9.1442,Z 133,A 171.7384,B 24.9553,C -1.5449,E1 24.8403,E2 274.612} C_DIS
LIN {X -124.2394,Y 12.5574,Z 133,A 170.2048,B 24.9549,C -1.5517,E1 24.8407,E2 276.1386} C_DIS
LIN {X -123.9788,Y 14.8927,Z 133,A 169.0634,B 24.9549,C -1.5525,E1 24.8411,E2 277.2849} C_DIS
LIN {X -123.5332,Y 18.2397,Z 133,A 167.5524,B 24.9544,C -1.5593,E1 24.8417,E2 278.7889} C_DIS
LIN {X -123.1574,Y 20.6093,Z 133,A 166.3998,B 24.9544,C -1.5606,E1 24.8422,E2 279.9452} C_DIS
LIN {X -122.5658,Y 23.8834,Z 133,A 164.9414,B 24.9539,C -1.5686,E1 24.8429,E2 281.3932} C_DIS
LIN {X -122.0238,Y 26.5091,Z 133,A 163.653,B 24.9539,C -1.57,E1 24.8437,E2 282.6857} C_DIS
LIN {X -121.3295,Y 29.5249,Z 133,A 162.2088,B 24.9536,C -1.5735,E1 24.8446,E2 284.13} C_DIS
LIN {X -120.4762,Y 32.8428,Z 133,A 160.6426,B 24.9533,C -1.5788,E1 24.8457,E2 285.6928} C_DIS
LIN {X -119.7402,Y 35.4239,Z 133,A 159.4132,B 24.9531,C -1.5829,E1 24.8467,E2 286.9196} C_DIS
LIN {X -118.8421,Y 38.3307,Z 133,A 157.9608,B 24.9529,C -1.5848,E1 24.8479,E2 288.3757} C_DIS
LIN {X -117.7477,Y 41.5771,Z 133,A 156.4184,B 24.9526,C -1.5911,E1 24.8493,E2 289.912} C_DIS
Enddeposition()
END
